LIN {X -15.999,Y -33.308,Z -148.499,A -90.000,B 90.000,C 0.000} C_DIS
LIN {X -18.536,Y -33.308,Z -146.844,A -90.000,B 90.000,C 0.000} C_DIS
LIN {X -19.606,Y -33.308,Z -146.164,A -90.000,B 90.000,C 0.000} C_DIS
LIN {X -20.856,Y -33.308,Z -145.200,A -90.000,B 90.000,C 0.000} C_DIS
LIN {X -22.809,Y -33.308,Z -143.742,A -90.000,B 90.000,C 0.000} C_DIS
LIN {X -23.151,Y -33.308,Z -143.479,A -90.000,B 90.000,C 0.000} C_DIS
LIN {X -23.524,Y -33.308,Z -143.181,A -90.000,B 90.000,C 0.000} C_DIS
LIN {X -25.307,Y -33.308,Z -141.556,A -90.000,B 90.000,C 0.000} C_DIS
LIN {X -26.828,Y -33.308,Z -140.210,A -90.000,B 90.000,C 0.000} C_DIS
LIN {X -27.168,Y -33.308,Z -139.876,A -90.000,B 90.000,C 0.000} C_DIS
LIN {X -27.524,Y -33.308,Z -139.495,A -90.000,B 90.000,C 0.000} C_DIS
LIN {X -28.033,Y -33.308,Z -138.967,A -90.000,B 90.000,C 0.000} C_DIS
LIN {X -30.108,Y -33.308,Z -136.726,A -90.000,B 90.000,C 0.000} C_DIS
LIN {X -30.362,Y -33.308,Z -136.404,A -90.000,B 90.000,C 0.000} C_DIS
LIN {X -31.175,Y -33.308,Z -135.330,A -90.000,B 90.000,C 0.000} C_DIS
LIN {X -32.732,Y -33.308,Z -133.288,A -90.000,B 90.000,C 0.000} C_DIS
LIN {X -32.993,Y -33.308,Z -132.891,A -90.000,B 90.000,C 0.000} C_DIS
LIN {X -34.951,Y -33.308,Z -129.675,A -90.000,B 90.000,C 0.000} C_DIS
LIN {X -35.160,Y -33.308,Z -129.243,A -90.000,B 90.000,C 0.000} C_DIS
LIN {X -36.562,Y -33.308,Z -126.281,A -90.000,B 90.000,C 0.000} C_DIS
LIN {X -36.636,Y -33.308,Z -126.118,A -90.000,B 90.000,C 0.000} C_DIS
LIN {X -37.764,Y -33.308,Z -123.048,A -90.000,B 90.000,C 0.000} C_DIS
LIN {X -37.875,Y -33.308,Z -122.732,A -90.000,B 90.000,C 0.000} C_DIS
LIN {X -37.915,Y -33.308,Z -122.610,A -90.000,B 90.000,C 0.000} C_DIS
LIN {X -38.201,Y -33.308,Z -121.561,A -90.000,B 90.000,C 0.000} C_DIS
LIN {X -38.605,Y -33.308,Z -120.049,A -90.000,B 90.000,C 0.000} C_DIS
LIN {X -38.751,Y -33.308,Z -119.515,A -90.000,B 90.000,C 0.000} C_DIS
LIN {X -38.857,Y -33.308,Z -119.060,A -90.000,B 90.000,C 0.000} C_DIS
LIN {X -39.050,Y -33.308,Z -118.006,A -90.000,B 90.000,C 0.000} C_DIS
LIN {X -39.335,Y -33.308,Z -116.504,A -90.000,B 90.000,C 0.000} C_DIS
LIN {X -39.510,Y -33.308,Z -115.571,A -90.000,B 90.000,C 0.000} C_DIS
LIN {X -39.533,Y -33.308,Z -115.382,A -90.000,B 90.000,C 0.000} C_DIS
LIN {X -39.662,Y -33.308,Z -114.053,A -90.000,B 90.000,C 0.000} C_DIS
LIN {X -39.769,Y -33.308,Z -112.841,A -90.000,B 90.000,C 0.000} C_DIS
LIN {X -39.851,Y -33.308,Z -111.994,A -90.000,B 90.000,C 0.000} C_DIS
LIN {X -39.881,Y -33.308,Z -111.571,A -90.000,B 90.000,C 0.000} C_DIS
LIN {X -39.882,Y -33.308,Z -111.344,A -90.000,B 90.000,C 0.000} C_DIS
LIN {X -39.887,Y -33.308,Z -111.029,A -90.000,B 90.000,C 0.000} C_DIS
LIN {X -39.893,Y -33.308,Z -109.551,A -90.000,B 90.000,C 0.000} C_DIS
LIN {X -39.909,Y -33.308,Z -108.367,A -90.000,B 90.000,C 0.000} C_DIS
LIN {X -39.903,Y -33.308,Z -107.912,A -90.000,B 90.000,C 0.000} C_DIS
LIN {X -39.874,Y -33.308,Z -107.539,A -90.000,B 90.000,C 0.000} C_DIS
LIN {X -39.834,Y -33.308,Z -106.670,A -90.000,B 90.000,C 0.000} C_DIS
LIN {X -39.843,Y -33.308,Z -106.632,A -90.000,B 90.000,C 0.000} C_DIS
LIN {X -40.216,Y -33.308,Z -105.871,A -90.000,B 90.000,C 0.000} C_DIS
LIN {X -40.541,Y -33.308,Z -105.425,A -90.000,B 90.000,C 0.000} C_DIS
LIN {X -41.279,Y -33.308,Z -104.304,A -90.000,B 90.000,C 0.000} C_DIS
LIN {X -41.681,Y -33.308,Z -103.742,A -90.000,B 90.000,C 0.000} C_DIS
LIN {X -42.580,Y -33.308,Z -102.613,A -90.000,B 90.000,C 0.000} C_DIS
LIN {X -42.846,Y -33.308,Z -102.253,A -90.000,B 90.000,C 0.000} C_DIS
LIN {X -43.563,Y -33.308,Z -101.346,A -90.000,B 90.000,C 0.000} C_DIS
LIN {X -44.397,Y -33.308,Z -100.200,A -90.000,B 90.000,C 0.000} C_DIS
LIN {X -44.716,Y -33.308,Z -99.731,A -90.000,B 90.000,C 0.000} C_DIS
LIN {X -45.686,Y -33.308,Z -98.284,A -90.000,B 90.000,C 0.000} C_DIS
LIN {X -46.185,Y -33.308,Z -97.544,A -90.000,B 90.000,C 0.000} C_DIS
LIN {X -46.405,Y -33.308,Z -97.201,A -90.000,B 90.000,C 0.000} C_DIS
LIN {X -46.712,Y -33.308,Z -96.706,A -90.000,B 90.000,C 0.000} C_DIS
LIN {X -47.443,Y -33.308,Z -95.513,A -90.000,B 90.000,C 0.000} C_DIS
LIN {X -47.884,Y -33.308,Z -94.789,A -90.000,B 90.000,C 0.000} C_DIS
LIN {X -48.028,Y -33.308,Z -94.546,A -90.000,B 90.000,C 0.000} C_DIS
LIN {X -48.144,Y -33.308,Z -94.332,A -90.000,B 90.000,C 0.000} C_DIS
LIN {X -48.227,Y -33.308,Z -94.169,A -90.000,B 90.000,C 0.000} C_DIS
LIN {X -49.715,Y -33.308,Z -90.825,A -90.000,B 90.000,C 0.000} C_DIS
LIN {X -49.898,Y -33.308,Z -90.362,A -90.000,B 90.000,C 0.000} C_DIS
LIN {X -50.066,Y -33.308,Z -89.882,A -90.000,B 90.000,C 0.000} C_DIS
LIN {X -50.156,Y -33.308,Z -89.607,A -90.000,B 90.000,C 0.000} C_DIS
LIN {X -50.572,Y -33.308,Z -88.253,A -90.000,B 90.000,C 0.000} C_DIS
LIN {X -50.836,Y -33.308,Z -87.423,A -90.000,B 90.000,C 0.000} C_DIS
LIN {X -51.046,Y -33.308,Z -86.747,A -90.000,B 90.000,C 0.000} C_DIS
LIN {X -51.153,Y -33.308,Z -86.380,A -90.000,B 90.000,C 0.000} C_DIS
LIN {X -51.746,Y -33.308,Z -84.240,A -90.000,B 90.000,C 0.000} C_DIS
LIN {X -52.221,Y -33.308,Z -82.065,A -90.000,B 90.000,C 0.000} C_DIS
LIN {X -52.576,Y -33.308,Z -80.127,A -90.000,B 90.000,C 0.000} C_DIS
LIN {X -52.615,Y -33.308,Z -79.847,A -90.000,B 90.000,C 0.000} C_DIS
LIN {X -52.708,Y -33.308,Z -78.854,A -90.000,B 90.000,C 0.000} C_DIS
LIN {X -52.791,Y -33.308,Z -78.084,A -90.000,B 90.000,C 0.000} C_DIS
LIN {X -52.824,Y -33.308,Z -76.672,A -90.000,B 90.000,C 0.000} C_DIS
LIN {X -52.824,Y -33.308,Z -76.379,A -90.000,B 90.000,C 0.000} C_DIS
LIN {X -52.821,Y -33.308,Z -76.293,A -90.000,B 90.000,C 0.000} C_DIS
LIN {X -52.840,Y -33.308,Z -76.082,A -90.000,B 90.000,C 0.000} C_DIS
LIN {X -52.839,Y -33.308,Z -74.765,A -90.000,B 90.000,C 0.000} C_DIS
LIN {X -52.858,Y -33.308,Z -74.482,A -90.000,B 90.000,C 0.000} C_DIS
LIN {X -52.768,Y -33.308,Z -73.356,A -90.000,B 90.000,C 0.000} C_DIS
LIN {X -52.777,Y -33.308,Z -72.948,A -90.000,B 90.000,C 0.000} C_DIS
LIN {X -52.757,Y -33.308,Z -72.712,A -90.000,B 90.000,C 0.000} C_DIS
LIN {X -52.602,Y -33.308,Z -71.811,A -90.000,B 90.000,C 0.000} C_DIS
LIN {X -52.589,Y -33.308,Z -71.493,A -90.000,B 90.000,C 0.000} C_DIS
LIN {X -52.569,Y -33.308,Z -71.257,A -90.000,B 90.000,C 0.000} C_DIS
LIN {X -52.319,Y -33.308,Z -70.370,A -90.000,B 90.000,C 0.000} C_DIS
LIN {X -52.254,Y -33.308,Z -69.902,A -90.000,B 90.000,C 0.000} C_DIS
LIN {X -52.185,Y -33.308,Z -69.675,A -90.000,B 90.000,C 0.000} C_DIS
LIN {X -51.762,Y -33.308,Z -68.858,A -90.000,B 90.000,C 0.000} C_DIS
LIN {X -51.636,Y -33.308,Z -68.514,A -90.000,B 90.000,C 0.000} C_DIS
LIN {X -51.589,Y -33.308,Z -68.423,A -90.000,B 90.000,C 0.000} C_DIS
LIN {X -51.480,Y -33.308,Z -68.226,A -90.000,B 90.000,C 0.000} C_DIS
LIN {X -51.476,Y -33.308,Z -68.222,A -90.000,B 90.000,C 0.000} C_DIS
LIN {X -51.325,Y -33.308,Z -68.048,A -90.000,B 90.000,C 0.000} C_DIS
LIN {X -50.280,Y -33.308,Z -66.958,A -90.000,B 90.000,C 0.000} C_DIS
LIN {X -50.251,Y -33.308,Z -66.924,A -90.000,B 90.000,C 0.000} C_DIS
LIN {X -50.061,Y -33.308,Z -66.782,A -90.000,B 90.000,C 0.000} C_DIS
LIN {X -50.009,Y -33.308,Z -66.752,A -90.000,B 90.000,C 0.000} C_DIS
LIN {X -49.012,Y -33.308,Z -66.062,A -90.000,B 90.000,C 0.000} C_DIS
LIN {X -48.527,Y -33.308,Z -65.766,A -90.000,B 90.000,C 0.000} C_DIS
LIN {X -48.102,Y -33.308,Z -65.546,A -90.000,B 90.000,C 0.000} C_DIS
LIN {X -47.850,Y -33.308,Z -65.419,A -90.000,B 90.000,C 0.000} C_DIS
LIN {X -46.602,Y -33.308,Z -64.968,A -90.000,B 90.000,C 0.000} C_DIS
LIN {X -45.421,Y -33.308,Z -64.531,A -90.000,B 90.000,C 0.000} C_DIS
LIN {X -45.151,Y -33.308,Z -64.451,A -90.000,B 90.000,C 0.000} C_DIS
LIN {X -44.503,Y -33.308,Z -64.272,A -90.000,B 90.000,C 0.000} C_DIS
LIN {X -43.209,Y -33.308,Z -63.965,A -90.000,B 90.000,C 0.000} C_DIS
LIN {X -43.095,Y -33.308,Z -63.939,A -90.000,B 90.000,C 0.000} C_DIS
LIN {X -40.860,Y -33.308,Z -63.512,A -90.000,B 90.000,C 0.000} C_DIS
LIN {X -40.000,Y -33.308,Z -63.408,A -90.000,B 90.000,C 0.000} C_DIS
LIN {X -39.681,Y -33.308,Z -63.385,A -90.000,B 90.000,C 0.000} C_DIS
LIN {X -39.254,Y -33.308,Z -63.373,A -90.000,B 90.000,C 0.000} C_DIS
LIN {X -36.732,Y -33.308,Z -63.251,A -90.000,B 90.000,C 0.000} C_DIS
LIN {X -35.728,Y -33.308,Z -63.273,A -90.000,B 90.000,C 0.000} C_DIS
LIN {X -35.378,Y -33.308,Z -63.300,A -90.000,B 90.000,C 0.000} C_DIS
LIN {X -33.474,Y -33.308,Z -63.465,A -90.000,B 90.000,C 0.000} C_DIS
LIN {X -33.246,Y -33.308,Z -63.489,A -90.000,B 90.000,C 0.000} C_DIS
LIN {X -32.432,Y -33.308,Z -63.617,A -90.000,B 90.000,C 0.000} C_DIS
LIN {X -30.767,Y -33.308,Z -63.887,A -90.000,B 90.000,C 0.000} C_DIS
LIN {X -30.545,Y -33.308,Z -63.929,A -90.000,B 90.000,C 0.000} C_DIS
LIN {X -30.194,Y -33.308,Z -63.999,A -90.000,B 90.000,C 0.000} C_DIS
LIN {X -28.705,Y -33.308,Z -64.309,A -90.000,B 90.000,C 0.000} C_DIS
LIN {X -28.123,Y -33.308,Z -64.436,A -90.000,B 90.000,C 0.000} C_DIS
LIN {X -28.013,Y -33.308,Z -64.462,A -90.000,B 90.000,C 0.000} C_DIS
LIN {X -25.914,Y -33.308,Z -65.027,A -90.000,B 90.000,C 0.000} C_DIS
LIN {X -24.380,Y -33.308,Z -65.532,A -90.000,B 90.000,C 0.000} C_DIS
LIN {X -24.132,Y -33.308,Z -65.610,A -90.000,B 90.000,C 0.000} C_DIS
LIN {X -23.744,Y -33.308,Z -65.739,A -90.000,B 90.000,C 0.000} C_DIS
LIN {X -22.588,Y -33.308,Z -66.146,A -90.000,B 90.000,C 0.000} C_DIS
LIN {X -21.576,Y -33.308,Z -66.458,A -90.000,B 90.000,C 0.000} C_DIS
LIN {X -21.536,Y -33.308,Z -66.468,A -90.000,B 90.000,C 0.000} C_DIS
LIN {X -21.279,Y -33.308,Z -65.952,A -90.000,B 90.000,C 0.000} C_DIS
LIN {X -21.202,Y -33.308,Z -65.724,A -90.000,B 90.000,C 0.000} C_DIS
LIN {X -20.968,Y -33.308,Z -65.093,A -90.000,B 90.000,C 0.000} C_DIS
LIN {X -20.909,Y -33.308,Z -64.895,A -90.000,B 90.000,C 0.000} C_DIS
LIN {X -20.659,Y -33.308,Z -64.202,A -90.000,B 90.000,C 0.000} C_DIS
LIN {X -20.533,Y -33.308,Z -63.908,A -90.000,B 90.000,C 0.000} C_DIS
LIN {X -20.359,Y -33.308,Z -63.600,A -90.000,B 90.000,C 0.000} C_DIS
LIN {X -20.270,Y -33.308,Z -63.460,A -90.000,B 90.000,C 0.000} C_DIS
LIN {X -19.954,Y -33.308,Z -62.911,A -90.000,B 90.000,C 0.000} C_DIS
LIN {X -19.740,Y -33.308,Z -62.631,A -90.000,B 90.000,C 0.000} C_DIS
LIN {X -19.479,Y -33.308,Z -62.376,A -90.000,B 90.000,C 0.000} C_DIS
LIN {X -19.448,Y -33.308,Z -62.349,A -90.000,B 90.000,C 0.000} C_DIS
LIN {X -19.165,Y -33.308,Z -62.141,A -90.000,B 90.000,C 0.000} C_DIS
LIN {X -18.817,Y -33.308,Z -61.902,A -90.000,B 90.000,C 0.000} C_DIS
LIN {X -18.540,Y -33.308,Z -61.737,A -90.000,B 90.000,C 0.000} C_DIS
LIN {X -18.265,Y -33.308,Z -61.626,A -90.000,B 90.000,C 0.000} C_DIS
LIN {X -17.942,Y -33.308,Z -61.498,A -90.000,B 90.000,C 0.000} C_DIS
LIN {X -17.612,Y -33.308,Z -61.377,A -90.000,B 90.000,C 0.000} C_DIS
LIN {X -16.997,Y -33.308,Z -61.181,A -90.000,B 90.000,C 0.000} C_DIS
LIN {X -16.111,Y -33.308,Z -60.930,A -90.000,B 90.000,C 0.000} C_DIS
LIN {X -15.997,Y -33.308,Z -60.903,A -90.000,B 90.000,C 0.000} C_DIS
LIN {X -15.606,Y -33.308,Z -60.822,A -90.000,B 90.000,C 0.000} C_DIS
LIN {X -15.503,Y -33.308,Z -60.804,A -90.000,B 90.000,C 0.000} C_DIS
LIN {X -15.152,Y -33.308,Z -60.781,A -90.000,B 90.000,C 0.000} C_DIS
LIN {X -12.993,Y -33.308,Z -60.780,A -90.000,B 90.000,C 0.000} C_DIS
LIN {X -11.855,Y -33.308,Z -60.776,A -90.000,B 90.000,C 0.000} C_DIS
LIN {X -11.504,Y -33.308,Z -60.803,A -90.000,B 90.000,C 0.000} C_DIS
LIN {X -11.122,Y -33.308,Z -60.840,A -90.000,B 90.000,C 0.000} C_DIS
LIN {X -8.836,Y -33.308,Z -61.073,A -90.000,B 90.000,C 0.000} C_DIS
LIN {X -7.942,Y -33.308,Z -61.208,A -90.000,B 90.000,C 0.000} C_DIS
LIN {X -6.167,Y -33.308,Z -61.448,A -90.000,B 90.000,C 0.000} C_DIS
LIN {X -5.366,Y -33.308,Z -61.575,A -90.000,B 90.000,C 0.000} C_DIS
LIN {X -4.569,Y -33.308,Z -61.716,A -90.000,B 90.000,C 0.000} C_DIS
LIN {X -2.737,Y -33.308,Z -61.952,A -90.000,B 90.000,C 0.000} C_DIS
LIN {X -1.013,Y -33.308,Z -62.234,A -90.000,B 90.000,C 0.000} C_DIS
LIN {X 0.927,Y -33.308,Z -62.435,A -90.000,B 90.000,C 0.000} C_DIS
LIN {X 1.948,Y -33.308,Z -62.549,A -90.000,B 90.000,C 0.000} C_DIS
LIN {X 2.990,Y -33.308,Z -62.617,A -90.000,B 90.000,C 0.000} C_DIS
LIN {X 4.660,Y -33.308,Z -62.776,A -90.000,B 90.000,C 0.000} C_DIS
LIN {X 5.580,Y -33.308,Z -62.844,A -90.000,B 90.000,C 0.000} C_DIS
LIN {X 6.790,Y -33.308,Z -62.924,A -90.000,B 90.000,C 0.000} C_DIS
LIN {X 7.569,Y -33.308,Z -62.950,A -90.000,B 90.000,C 0.000} C_DIS
LIN {X 8.530,Y -33.308,Z -62.986,A -90.000,B 90.000,C 0.000} C_DIS
LIN {X 9.844,Y -33.308,Z -62.969,A -90.000,B 90.000,C 0.000} C_DIS
LIN {X 10.732,Y -33.308,Z -62.896,A -90.000,B 90.000,C 0.000} C_DIS
LIN {X 11.400,Y -33.308,Z -62.776,A -90.000,B 90.000,C 0.000} C_DIS
LIN {X 11.835,Y -33.308,Z -62.634,A -90.000,B 90.000,C 0.000} C_DIS
LIN {X 12.131,Y -33.308,Z -62.482,A -90.000,B 90.000,C 0.000} C_DIS
LIN {X 12.597,Y -33.308,Z -62.206,A -90.000,B 90.000,C 0.000} C_DIS
LIN {X 12.961,Y -33.308,Z -62.010,A -90.000,B 90.000,C 0.000} C_DIS
LIN {X 13.229,Y -33.308,Z -61.872,A -90.000,B 90.000,C 0.000} C_DIS
LIN {X 13.616,Y -33.308,Z -61.666,A -90.000,B 90.000,C 0.000} C_DIS
LIN {X 13.852,Y -33.308,Z -61.563,A -90.000,B 90.000,C 0.000} C_DIS
LIN {X 14.231,Y -33.308,Z -61.424,A -90.000,B 90.000,C 0.000} C_DIS
LIN {X 14.576,Y -33.308,Z -61.333,A -90.000,B 90.000,C 0.000} C_DIS
LIN {X 14.698,Y -33.308,Z -61.293,A -90.000,B 90.000,C 0.000} C_DIS
LIN {X 14.742,Y -33.308,Z -61.279,A -90.000,B 90.000,C 0.000} C_DIS
LIN {X 14.860,Y -33.308,Z -61.243,A -90.000,B 90.000,C 0.000} C_DIS
LIN {X 15.253,Y -33.308,Z -61.152,A -90.000,B 90.000,C 0.000} C_DIS
LIN {X 15.653,Y -33.308,Z -61.110,A -90.000,B 90.000,C 0.000} C_DIS
LIN {X 15.830,Y -33.308,Z -61.103,A -90.000,B 90.000,C 0.000} C_DIS
LIN {X 16.705,Y -33.308,Z -61.121,A -90.000,B 90.000,C 0.000} C_DIS
LIN {X 17.110,Y -33.308,Z -61.177,A -90.000,B 90.000,C 0.000} C_DIS
LIN {X 17.392,Y -33.308,Z -61.217,A -90.000,B 90.000,C 0.000} C_DIS
LIN {X 17.618,Y -33.308,Z -61.255,A -90.000,B 90.000,C 0.000} C_DIS
LIN {X 17.736,Y -33.308,Z -61.278,A -90.000,B 90.000,C 0.000} C_DIS
LIN {X 17.944,Y -33.308,Z -61.166,A -90.000,B 90.000,C 0.000} C_DIS
LIN {X 18.039,Y -33.308,Z -61.122,A -90.000,B 90.000,C 0.000} C_DIS
LIN {X 18.354,Y -33.308,Z -60.997,A -90.000,B 90.000,C 0.000} C_DIS
LIN {X 18.590,Y -33.308,Z -60.833,A -90.000,B 90.000,C 0.000} C_DIS
LIN {X 18.755,Y -33.308,Z -60.737,A -90.000,B 90.000,C 0.000} C_DIS
LIN {X 18.966,Y -33.308,Z -60.623,A -90.000,B 90.000,C 0.000} C_DIS
LIN {X 19.141,Y -33.308,Z -60.546,A -90.000,B 90.000,C 0.000} C_DIS
LIN {X 19.364,Y -33.308,Z -60.457,A -90.000,B 90.000,C 0.000} C_DIS
LIN {X 19.546,Y -33.308,Z -60.401,A -90.000,B 90.000,C 0.000} C_DIS
LIN {X 19.884,Y -33.308,Z -60.310,A -90.000,B 90.000,C 0.000} C_DIS
LIN {X 20.034,Y -33.308,Z -60.279,A -90.000,B 90.000,C 0.000} C_DIS
LIN {X 20.311,Y -33.308,Z -60.238,A -90.000,B 90.000,C 0.000} C_DIS
LIN {X 20.453,Y -33.308,Z -60.219,A -90.000,B 90.000,C 0.000} C_DIS
LIN {X 20.876,Y -33.308,Z -60.209,A -90.000,B 90.000,C 0.000} C_DIS
LIN {X 21.298,Y -33.308,Z -60.250,A -90.000,B 90.000,C 0.000} C_DIS
LIN {X 21.856,Y -33.308,Z -60.371,A -90.000,B 90.000,C 0.000} C_DIS
LIN {X 22.005,Y -33.308,Z -60.420,A -90.000,B 90.000,C 0.000} C_DIS
LIN {X 22.223,Y -33.308,Z -60.253,A -90.000,B 90.000,C 0.000} C_DIS
LIN {X 22.475,Y -33.308,Z -60.067,A -90.000,B 90.000,C 0.000} C_DIS
LIN {X 22.603,Y -33.308,Z -59.979,A -90.000,B 90.000,C 0.000} C_DIS
LIN {X 22.940,Y -33.308,Z -59.756,A -90.000,B 90.000,C 0.000} C_DIS
LIN {X 23.193,Y -33.308,Z -59.603,A -90.000,B 90.000,C 0.000} C_DIS
LIN {X 23.466,Y -33.308,Z -59.442,A -90.000,B 90.000,C 0.000} C_DIS
LIN {X 23.667,Y -33.308,Z -59.330,A -90.000,B 90.000,C 0.000} C_DIS
LIN {X 24.032,Y -33.308,Z -59.140,A -90.000,B 90.000,C 0.000} C_DIS
LIN {X 24.416,Y -33.308,Z -58.965,A -90.000,B 90.000,C 0.000} C_DIS
LIN {X 24.819,Y -33.308,Z -58.788,A -90.000,B 90.000,C 0.000} C_DIS
LIN {X 25.037,Y -33.308,Z -58.701,A -90.000,B 90.000,C 0.000} C_DIS
LIN {X 25.238,Y -33.308,Z -58.623,A -90.000,B 90.000,C 0.000} C_DIS
LIN {X 25.658,Y -33.308,Z -58.481,A -90.000,B 90.000,C 0.000} C_DIS
LIN {X 25.742,Y -33.308,Z -58.455,A -90.000,B 90.000,C 0.000} C_DIS
LIN {X 25.705,Y -33.308,Z -58.141,A -90.000,B 90.000,C 0.000} C_DIS
LIN {X 25.684,Y -33.308,Z -57.920,A -90.000,B 90.000,C 0.000} C_DIS
LIN {X 25.655,Y -33.308,Z -57.445,A -90.000,B 90.000,C 0.000} C_DIS
LIN {X 25.677,Y -33.308,Z -56.969,A -90.000,B 90.000,C 0.000} C_DIS
LIN {X 25.730,Y -33.308,Z -56.579,A -90.000,B 90.000,C 0.000} C_DIS
LIN {X 25.823,Y -33.308,Z -56.121,A -90.000,B 90.000,C 0.000} C_DIS
LIN {X 25.964,Y -33.308,Z -55.675,A -90.000,B 90.000,C 0.000} C_DIS
LIN {X 26.151,Y -33.308,Z -55.247,A -90.000,B 90.000,C 0.000} C_DIS
LIN {X 26.465,Y -33.308,Z -54.700,A -90.000,B 90.000,C 0.000} C_DIS
LIN {X 26.502,Y -33.308,Z -54.645,A -90.000,B 90.000,C 0.000} C_DIS
LIN {X 26.706,Y -33.308,Z -54.362,A -90.000,B 90.000,C 0.000} C_DIS
LIN {X 26.778,Y -33.308,Z -54.272,A -90.000,B 90.000,C 0.000} C_DIS
LIN {X 27.012,Y -33.308,Z -54.013,A -90.000,B 90.000,C 0.000} C_DIS
LIN {X 27.093,Y -33.308,Z -53.931,A -90.000,B 90.000,C 0.000} C_DIS
LIN {X 27.353,Y -33.308,Z -53.699,A -90.000,B 90.000,C 0.000} C_DIS
LIN {X 27.443,Y -33.308,Z -53.626,A -90.000,B 90.000,C 0.000} C_DIS
LIN {X 27.726,Y -33.308,Z -53.423,A -90.000,B 90.000,C 0.000} C_DIS
LIN {X 27.823,Y -33.308,Z -53.360,A -90.000,B 90.000,C 0.000} C_DIS
LIN {X 28.127,Y -33.308,Z -53.188,A -90.000,B 90.000,C 0.000} C_DIS
LIN {X 28.289,Y -33.308,Z -53.103,A -90.000,B 90.000,C 0.000} C_DIS
LIN {X 28.423,Y -33.308,Z -53.037,A -90.000,B 90.000,C 0.000} C_DIS
LIN {X 28.711,Y -33.308,Z -52.912,A -90.000,B 90.000,C 0.000} C_DIS
LIN {X 28.851,Y -33.308,Z -52.861,A -90.000,B 90.000,C 0.000} C_DIS
LIN {X 29.151,Y -33.308,Z -52.767,A -90.000,B 90.000,C 0.000} C_DIS
LIN {X 29.219,Y -33.308,Z -52.748,A -90.000,B 90.000,C 0.000} C_DIS
LIN {X 29.223,Y -33.308,Z -52.612,A -90.000,B 90.000,C 0.000} C_DIS
LIN {X 29.286,Y -33.308,Z -52.163,A -90.000,B 90.000,C 0.000} C_DIS
LIN {X 29.356,Y -33.308,Z -51.864,A -90.000,B 90.000,C 0.000} C_DIS
LIN {X 29.424,Y -33.308,Z -51.550,A -90.000,B 90.000,C 0.000} C_DIS
LIN {X 29.529,Y -33.308,Z -51.140,A -90.000,B 90.000,C 0.000} C_DIS
LIN {X 29.681,Y -33.308,Z -50.745,A -90.000,B 90.000,C 0.000} C_DIS
LIN {X 29.756,Y -33.308,Z -50.567,A -90.000,B 90.000,C 0.000} C_DIS
LIN {X 29.940,Y -33.308,Z -50.168,A -90.000,B 90.000,C 0.000} C_DIS
LIN {X 30.138,Y -33.308,Z -49.793,A -90.000,B 90.000,C 0.000} C_DIS
LIN {X 30.158,Y -33.308,Z -49.758,A -90.000,B 90.000,C 0.000} C_DIS
LIN {X 30.387,Y -33.308,Z -49.416,A -90.000,B 90.000,C 0.000} C_DIS
LIN {X 30.427,Y -33.308,Z -49.361,A -90.000,B 90.000,C 0.000} C_DIS
LIN {X 30.699,Y -33.308,Z -48.997,A -90.000,B 90.000,C 0.000} C_DIS
LIN {X 30.764,Y -33.308,Z -48.903,A -90.000,B 90.000,C 0.000} C_DIS
LIN {X 30.798,Y -33.308,Z -48.858,A -90.000,B 90.000,C 0.000} C_DIS
LIN {X 31.083,Y -33.308,Z -48.522,A -90.000,B 90.000,C 0.000} C_DIS
LIN {X 31.405,Y -33.308,Z -48.220,A -90.000,B 90.000,C 0.000} C_DIS
LIN {X 31.941,Y -33.308,Z -47.791,A -90.000,B 90.000,C 0.000} C_DIS
LIN {X 31.970,Y -33.308,Z -47.764,A -90.000,B 90.000,C 0.000} C_DIS
LIN {X 32.324,Y -33.308,Z -47.500,A -90.000,B 90.000,C 0.000} C_DIS
LIN {X 32.717,Y -33.308,Z -47.272,A -90.000,B 90.000,C 0.000} C_DIS
LIN {X 32.794,Y -33.308,Z -47.233,A -90.000,B 90.000,C 0.000} C_DIS
LIN {X 33.121,Y -33.308,Z -47.090,A -90.000,B 90.000,C 0.000} C_DIS
LIN {X 33.449,Y -33.308,Z -46.955,A -90.000,B 90.000,C 0.000} C_DIS
LIN {X 33.884,Y -33.308,Z -46.784,A -90.000,B 90.000,C 0.000} C_DIS
LIN {X 34.311,Y -33.308,Z -46.652,A -90.000,B 90.000,C 0.000} C_DIS
LIN {X 34.813,Y -33.308,Z -46.529,A -90.000,B 90.000,C 0.000} C_DIS
LIN {X 35.264,Y -33.308,Z -46.469,A -90.000,B 90.000,C 0.000} C_DIS
LIN {X 35.688,Y -33.308,Z -46.434,A -90.000,B 90.000,C 0.000} C_DIS
LIN {X 36.302,Y -33.308,Z -46.365,A -90.000,B 90.000,C 0.000} C_DIS
LIN {X 36.835,Y -33.308,Z -46.338,A -90.000,B 90.000,C 0.000} C_DIS
LIN {X 37.302,Y -33.308,Z -46.347,A -90.000,B 90.000,C 0.000} C_DIS
LIN {X 37.688,Y -33.308,Z -46.382,A -90.000,B 90.000,C 0.000} C_DIS
LIN {X 38.275,Y -33.308,Z -46.449,A -90.000,B 90.000,C 0.000} C_DIS
LIN {X 38.738,Y -33.308,Z -46.508,A -90.000,B 90.000,C 0.000} C_DIS
LIN {X 39.091,Y -33.308,Z -46.568,A -90.000,B 90.000,C 0.000} C_DIS
LIN {X 40.567,Y -33.308,Z -46.891,A -90.000,B 90.000,C 0.000} C_DIS
LIN {X 41.529,Y -33.308,Z -47.060,A -90.000,B 90.000,C 0.000} C_DIS
LIN {X 42.172,Y -33.308,Z -47.093,A -90.000,B 90.000,C 0.000} C_DIS
LIN {X 43.024,Y -33.308,Z -46.949,A -90.000,B 90.000,C 0.000} C_DIS
LIN {X 43.517,Y -33.308,Z -46.826,A -90.000,B 90.000,C 0.000} C_DIS
LIN {X 44.454,Y -33.308,Z -46.576,A -90.000,B 90.000,C 0.000} C_DIS
LIN {X 45.621,Y -33.308,Z -46.357,A -90.000,B 90.000,C 0.000} C_DIS
LIN {X 46.224,Y -33.308,Z -46.219,A -90.000,B 90.000,C 0.000} C_DIS
LIN {X 46.763,Y -33.308,Z -46.136,A -90.000,B 90.000,C 0.000} C_DIS
LIN {X 47.215,Y -33.308,Z -46.104,A -90.000,B 90.000,C 0.000} C_DIS
LIN {X 47.811,Y -33.308,Z -46.089,A -90.000,B 90.000,C 0.000} C_DIS
LIN {X 48.729,Y -33.308,Z -46.110,A -90.000,B 90.000,C 0.000} C_DIS
LIN {X 49.207,Y -33.308,Z -46.147,A -90.000,B 90.000,C 0.000} C_DIS
LIN {X 49.600,Y -33.308,Z -46.184,A -90.000,B 90.000,C 0.000} C_DIS
LIN {X 50.226,Y -33.308,Z -46.292,A -90.000,B 90.000,C 0.000} C_DIS
LIN {X 50.651,Y -33.308,Z -46.408,A -90.000,B 90.000,C 0.000} C_DIS
LIN {X 51.282,Y -33.308,Z -46.611,A -90.000,B 90.000,C 0.000} C_DIS
LIN {X 52.189,Y -33.308,Z -46.925,A -90.000,B 90.000,C 0.000} C_DIS
LIN {X 53.231,Y -33.308,Z -47.364,A -90.000,B 90.000,C 0.000} C_DIS
LIN {X 53.647,Y -33.308,Z -47.549,A -90.000,B 90.000,C 0.000} C_DIS
LIN {X 54.040,Y -33.308,Z -47.779,A -90.000,B 90.000,C 0.000} C_DIS
LIN {X 56.196,Y -33.308,Z -49.211,A -90.000,B 90.000,C 0.000} C_DIS
LIN {X 56.730,Y -33.308,Z -49.569,A -90.000,B 90.000,C 0.000} C_DIS
LIN {X 57.096,Y -33.308,Z -49.840,A -90.000,B 90.000,C 0.000} C_DIS
LIN {X 59.476,Y -33.308,Z -51.862,A -90.000,B 90.000,C 0.000} C_DIS
LIN {X 59.810,Y -33.308,Z -52.171,A -90.000,B 90.000,C 0.000} C_DIS
LIN {X 62.039,Y -33.308,Z -54.281,A -90.000,B 90.000,C 0.000} C_DIS
LIN {X 63.618,Y -33.308,Z -55.808,A -90.000,B 90.000,C 0.000} C_DIS
LIN {X 64.198,Y -33.308,Z -56.378,A -90.000,B 90.000,C 0.000} C_DIS
LIN {X 64.715,Y -33.308,Z -56.862,A -90.000,B 90.000,C 0.000} C_DIS
LIN {X 66.205,Y -33.308,Z -58.228,A -90.000,B 90.000,C 0.000} C_DIS
LIN {X 68.301,Y -33.308,Z -60.193,A -90.000,B 90.000,C 0.000} C_DIS
LIN {X 69.366,Y -33.308,Z -61.311,A -90.000,B 90.000,C 0.000} C_DIS
LIN {X 70.233,Y -33.308,Z -62.330,A -90.000,B 90.000,C 0.000} C_DIS
LIN {X 71.735,Y -33.308,Z -64.192,A -90.000,B 90.000,C 0.000} C_DIS
LIN {X 71.839,Y -33.308,Z -64.323,A -90.000,B 90.000,C 0.000} C_DIS
LIN {X 72.046,Y -33.308,Z -64.596,A -90.000,B 90.000,C 0.000} C_DIS
LIN {X 72.489,Y -33.308,Z -65.199,A -90.000,B 90.000,C 0.000} C_DIS
LIN {X 72.909,Y -33.308,Z -65.812,A -90.000,B 90.000,C 0.000} C_DIS
LIN {X 73.188,Y -33.308,Z -66.158,A -90.000,B 90.000,C 0.000} C_DIS
LIN {X 73.389,Y -33.308,Z -66.438,A -90.000,B 90.000,C 0.000} C_DIS
LIN {X 73.517,Y -33.308,Z -66.628,A -90.000,B 90.000,C 0.000} C_DIS
LIN {X 73.829,Y -33.308,Z -67.008,A -90.000,B 90.000,C 0.000} C_DIS
LIN {X 74.218,Y -33.308,Z -67.509,A -90.000,B 90.000,C 0.000} C_DIS
LIN {X 74.278,Y -33.308,Z -67.577,A -90.000,B 90.000,C 0.000} C_DIS
LIN {X 74.534,Y -33.308,Z -67.914,A -90.000,B 90.000,C 0.000} C_DIS
LIN {X 74.861,Y -33.308,Z -68.353,A -90.000,B 90.000,C 0.000} C_DIS
LIN {X 75.321,Y -33.308,Z -68.845,A -90.000,B 90.000,C 0.000} C_DIS
LIN {X 75.520,Y -33.308,Z -69.107,A -90.000,B 90.000,C 0.000} C_DIS
LIN {X 76.204,Y -33.308,Z -69.865,A -90.000,B 90.000,C 0.000} C_DIS
LIN {X 76.275,Y -33.308,Z -69.948,A -90.000,B 90.000,C 0.000} C_DIS
LIN {X 76.321,Y -33.308,Z -69.996,A -90.000,B 90.000,C 0.000} C_DIS
LIN {X 76.568,Y -33.308,Z -70.298,A -90.000,B 90.000,C 0.000} C_DIS
LIN {X 76.871,Y -33.308,Z -70.672,A -90.000,B 90.000,C 0.000} C_DIS
LIN {X 77.245,Y -33.308,Z -71.078,A -90.000,B 90.000,C 0.000} C_DIS
LIN {X 77.541,Y -33.308,Z -71.404,A -90.000,B 90.000,C 0.000} C_DIS
LIN {X 77.612,Y -33.308,Z -71.491,A -90.000,B 90.000,C 0.000} C_DIS
LIN {X 77.796,Y -33.308,Z -71.699,A -90.000,B 90.000,C 0.000} C_DIS
LIN {X 78.092,Y -33.308,Z -72.049,A -90.000,B 90.000,C 0.000} C_DIS
LIN {X 78.123,Y -33.308,Z -71.941,A -90.000,B 90.000,C 0.000} C_DIS
LIN {X 78.695,Y -33.308,Z -70.203,A -90.000,B 90.000,C 0.000} C_DIS
LIN {X 78.831,Y -33.308,Z -69.802,A -90.000,B 90.000,C 0.000} C_DIS
LIN {X 79.195,Y -33.308,Z -68.754,A -90.000,B 90.000,C 0.000} C_DIS
LIN {X 79.783,Y -33.308,Z -67.276,A -90.000,B 90.000,C 0.000} C_DIS
LIN {X 79.809,Y -33.308,Z -67.218,A -90.000,B 90.000,C 0.000} C_DIS
LIN {X 80.447,Y -33.308,Z -65.768,A -90.000,B 90.000,C 0.000} C_DIS
LIN {X 80.647,Y -33.308,Z -65.330,A -90.000,B 90.000,C 0.000} C_DIS
LIN {X 81.438,Y -33.308,Z -63.804,A -90.000,B 90.000,C 0.000} C_DIS
LIN {X 81.684,Y -33.308,Z -63.383,A -90.000,B 90.000,C 0.000} C_DIS
LIN {X 82.705,Y -33.308,Z -61.742,A -90.000,B 90.000,C 0.000} C_DIS
LIN {X 84.243,Y -33.308,Z -59.630,A -90.000,B 90.000,C 0.000} C_DIS
LIN {X 85.732,Y -33.308,Z -57.856,A -90.000,B 90.000,C 0.000} C_DIS
LIN {X 86.059,Y -33.308,Z -57.494,A -90.000,B 90.000,C 0.000} C_DIS
LIN {X 87.795,Y -33.308,Z -55.685,A -90.000,B 90.000,C 0.000} C_DIS
LIN {X 89.787,Y -33.308,Z -53.862,A -90.000,B 90.000,C 0.000} C_DIS
LIN {X 90.167,Y -33.308,Z -53.520,A -90.000,B 90.000,C 0.000} C_DIS
LIN {X 92.263,Y -33.308,Z -51.722,A -90.000,B 90.000,C 0.000} C_DIS
LIN {X 94.367,Y -33.308,Z -49.945,A -90.000,B 90.000,C 0.000} C_DIS
LIN {X 94.745,Y -33.308,Z -49.614,A -90.000,B 90.000,C 0.000} C_DIS
LIN {X 94.732,Y -33.308,Z -49.589,A -90.000,B 90.000,C 0.000} C_DIS
LIN {X 94.667,Y -33.308,Z -49.441,A -90.000,B 90.000,C 0.000} C_DIS
LIN {X 94.423,Y -33.308,Z -48.996,A -90.000,B 90.000,C 0.000} C_DIS
LIN {X 94.322,Y -33.308,Z -48.808,A -90.000,B 90.000,C 0.000} C_DIS
LIN {X 94.232,Y -33.308,Z -48.623,A -90.000,B 90.000,C 0.000} C_DIS
LIN {X 94.145,Y -33.308,Z -48.355,A -90.000,B 90.000,C 0.000} C_DIS
LIN {X 94.048,Y -33.308,Z -47.934,A -90.000,B 90.000,C 0.000} C_DIS
LIN {X 94.008,Y -33.308,Z -47.725,A -90.000,B 90.000,C 0.000} C_DIS
LIN {X 93.969,Y -33.308,Z -47.446,A -90.000,B 90.000,C 0.000} C_DIS
LIN {X 93.970,Y -33.308,Z -47.410,A -90.000,B 90.000,C 0.000} C_DIS
LIN {X 93.976,Y -33.308,Z -46.998,A -90.000,B 90.000,C 0.000} C_DIS
LIN {X 94.004,Y -33.308,Z -46.687,A -90.000,B 90.000,C 0.000} C_DIS
LIN {X 94.082,Y -33.308,Z -46.377,A -90.000,B 90.000,C 0.000} C_DIS
LIN {X 94.223,Y -33.308,Z -45.886,A -90.000,B 90.000,C 0.000} C_DIS
LIN {X 94.352,Y -33.308,Z -45.554,A -90.000,B 90.000,C 0.000} C_DIS
LIN {X 94.522,Y -33.308,Z -45.163,A -90.000,B 90.000,C 0.000} C_DIS
LIN {X 94.682,Y -33.308,Z -44.819,A -90.000,B 90.000,C 0.000} C_DIS
LIN {X 94.808,Y -33.308,Z -44.577,A -90.000,B 90.000,C 0.000} C_DIS
LIN {X 94.938,Y -33.308,Z -44.340,A -90.000,B 90.000,C 0.000} C_DIS
LIN {X 95.287,Y -33.308,Z -43.751,A -90.000,B 90.000,C 0.000} C_DIS
LIN {X 95.352,Y -33.308,Z -43.638,A -90.000,B 90.000,C 0.000} C_DIS
LIN {X 95.579,Y -33.308,Z -43.305,A -90.000,B 90.000,C 0.000} C_DIS
LIN {X 96.023,Y -33.308,Z -42.688,A -90.000,B 90.000,C 0.000} C_DIS
LIN {X 96.804,Y -33.308,Z -41.778,A -90.000,B 90.000,C 0.000} C_DIS
LIN {X 97.620,Y -33.308,Z -40.978,A -90.000,B 90.000,C 0.000} C_DIS
LIN {X 98.293,Y -33.308,Z -40.401,A -90.000,B 90.000,C 0.000} C_DIS
LIN {X 98.488,Y -33.308,Z -40.239,A -90.000,B 90.000,C 0.000} C_DIS
LIN {X 99.372,Y -33.308,Z -39.589,A -90.000,B 90.000,C 0.000} C_DIS
LIN {X 100.004,Y -33.308,Z -39.176,A -90.000,B 90.000,C 0.000} C_DIS
LIN {X 100.704,Y -33.308,Z -38.748,A -90.000,B 90.000,C 0.000} C_DIS
LIN {X 101.666,Y -33.308,Z -38.226,A -90.000,B 90.000,C 0.000} C_DIS
LIN {X 102.746,Y -33.308,Z -37.714,A -90.000,B 90.000,C 0.000} C_DIS
LIN {X 103.228,Y -33.308,Z -37.494,A -90.000,B 90.000,C 0.000} C_DIS
LIN {X 104.493,Y -33.308,Z -36.935,A -90.000,B 90.000,C 0.000} C_DIS
LIN {X 105.393,Y -33.308,Z -36.556,A -90.000,B 90.000,C 0.000} C_DIS
LIN {X 106.867,Y -33.308,Z -35.970,A -90.000,B 90.000,C 0.000} C_DIS
LIN {X 107.391,Y -33.308,Z -35.771,A -90.000,B 90.000,C 0.000} C_DIS
LIN {X 107.871,Y -33.308,Z -35.598,A -90.000,B 90.000,C 0.000} C_DIS
LIN {X 108.337,Y -33.308,Z -35.443,A -90.000,B 90.000,C 0.000} C_DIS
LIN {X 108.769,Y -33.308,Z -35.328,A -90.000,B 90.000,C 0.000} C_DIS
LIN {X 109.226,Y -33.308,Z -35.225,A -90.000,B 90.000,C 0.000} C_DIS
LIN {X 109.649,Y -33.308,Z -35.169,A -90.000,B 90.000,C 0.000} C_DIS
LIN {X 110.108,Y -33.308,Z -35.113,A -90.000,B 90.000,C 0.000} C_DIS
LIN {X 110.614,Y -33.308,Z -35.106,A -90.000,B 90.000,C 0.000} C_DIS
LIN {X 110.969,Y -33.308,Z -35.118,A -90.000,B 90.000,C 0.000} C_DIS
LIN {X 111.443,Y -33.308,Z -35.160,A -90.000,B 90.000,C 0.000} C_DIS
LIN {X 112.073,Y -33.308,Z -35.278,A -90.000,B 90.000,C 0.000} C_DIS
LIN {X 112.435,Y -33.308,Z -35.371,A -90.000,B 90.000,C 0.000} C_DIS
LIN {X 112.884,Y -33.308,Z -35.505,A -90.000,B 90.000,C 0.000} C_DIS
LIN {X 113.055,Y -33.308,Z -35.560,A -90.000,B 90.000,C 0.000} C_DIS
LIN {X 113.513,Y -33.308,Z -35.750,A -90.000,B 90.000,C 0.000} C_DIS
LIN {X 113.987,Y -33.308,Z -35.977,A -90.000,B 90.000,C 0.000} C_DIS
LIN {X 114.418,Y -33.308,Z -36.210,A -90.000,B 90.000,C 0.000} C_DIS
LIN {X 114.548,Y -33.308,Z -36.291,A -90.000,B 90.000,C 0.000} C_DIS
LIN {X 114.952,Y -33.308,Z -36.567,A -90.000,B 90.000,C 0.000} C_DIS
LIN {X 115.073,Y -33.308,Z -36.664,A -90.000,B 90.000,C 0.000} C_DIS
LIN {X 115.430,Y -33.308,Z -36.965,A -90.000,B 90.000,C 0.000} C_DIS
LIN {X 115.520,Y -33.308,Z -37.046,A -90.000,B 90.000,C 0.000} C_DIS
LIN {X 115.872,Y -33.308,Z -37.410,A -90.000,B 90.000,C 0.000} C_DIS
LIN {X 116.081,Y -33.308,Z -37.633,A -90.000,B 90.000,C 0.000} C_DIS
LIN {X 116.439,Y -33.308,Z -38.088,A -90.000,B 90.000,C 0.000} C_DIS
LIN {X 116.700,Y -33.308,Z -38.500,A -90.000,B 90.000,C 0.000} C_DIS
LIN {X 116.930,Y -33.308,Z -38.965,A -90.000,B 90.000,C 0.000} C_DIS
LIN {X 117.059,Y -33.308,Z -39.250,A -90.000,B 90.000,C 0.000} C_DIS
LIN {X 117.105,Y -33.308,Z -39.367,A -90.000,B 90.000,C 0.000} C_DIS
LIN {X 117.260,Y -33.308,Z -39.781,A -90.000,B 90.000,C 0.000} C_DIS
LIN {X 117.391,Y -33.308,Z -40.285,A -90.000,B 90.000,C 0.000} C_DIS
LIN {X 117.462,Y -33.308,Z -40.593,A -90.000,B 90.000,C 0.000} C_DIS
LIN {X 117.541,Y -33.308,Z -41.113,A -90.000,B 90.000,C 0.000} C_DIS
LIN {X 117.596,Y -33.308,Z -41.528,A -90.000,B 90.000,C 0.000} C_DIS
LIN {X 117.631,Y -33.308,Z -41.885,A -90.000,B 90.000,C 0.000} C_DIS
LIN {X 117.656,Y -33.308,Z -42.390,A -90.000,B 90.000,C 0.000} C_DIS
LIN {X 117.668,Y -33.308,Z -42.698,A -90.000,B 90.000,C 0.000} C_DIS
LIN {X 117.664,Y -33.308,Z -42.870,A -90.000,B 90.000,C 0.000} C_DIS
LIN {X 117.651,Y -33.308,Z -43.202,A -90.000,B 90.000,C 0.000} C_DIS
LIN {X 117.607,Y -33.308,Z -43.724,A -90.000,B 90.000,C 0.000} C_DIS
LIN {X 117.565,Y -33.308,Z -44.127,A -90.000,B 90.000,C 0.000} C_DIS
LIN {X 117.487,Y -33.308,Z -44.644,A -90.000,B 90.000,C 0.000} C_DIS
LIN {X 117.396,Y -33.308,Z -45.126,A -90.000,B 90.000,C 0.000} C_DIS
LIN {X 117.258,Y -33.308,Z -45.748,A -90.000,B 90.000,C 0.000} C_DIS
LIN {X 117.117,Y -33.308,Z -46.220,A -90.000,B 90.000,C 0.000} C_DIS
LIN {X 116.895,Y -33.308,Z -46.951,A -90.000,B 90.000,C 0.000} C_DIS
LIN {X 116.548,Y -33.308,Z -47.851,A -90.000,B 90.000,C 0.000} C_DIS
LIN {X 116.366,Y -33.308,Z -48.292,A -90.000,B 90.000,C 0.000} C_DIS
LIN {X 115.865,Y -33.308,Z -49.367,A -90.000,B 90.000,C 0.000} C_DIS
LIN {X 115.244,Y -33.308,Z -50.609,A -90.000,B 90.000,C 0.000} C_DIS
LIN {X 114.588,Y -33.308,Z -51.909,A -90.000,B 90.000,C 0.000} C_DIS
LIN {X 113.934,Y -33.308,Z -53.246,A -90.000,B 90.000,C 0.000} C_DIS
LIN {X 113.270,Y -33.308,Z -54.704,A -90.000,B 90.000,C 0.000} C_DIS
LIN {X 112.799,Y -33.308,Z -55.830,A -90.000,B 90.000,C 0.000} C_DIS
LIN {X 112.208,Y -33.308,Z -57.403,A -90.000,B 90.000,C 0.000} C_DIS
LIN {X 111.674,Y -33.308,Z -59.009,A -90.000,B 90.000,C 0.000} C_DIS
LIN {X 111.248,Y -33.308,Z -60.488,A -90.000,B 90.000,C 0.000} C_DIS
LIN {X 110.729,Y -33.308,Z -62.393,A -90.000,B 90.000,C 0.000} C_DIS
LIN {X 110.160,Y -33.308,Z -64.412,A -90.000,B 90.000,C 0.000} C_DIS
LIN {X 110.004,Y -33.308,Z -64.935,A -90.000,B 90.000,C 0.000} C_DIS
LIN {X 109.346,Y -33.308,Z -66.982,A -90.000,B 90.000,C 0.000} C_DIS
LIN {X 109.232,Y -33.308,Z -67.288,A -90.000,B 90.000,C 0.000} C_DIS
LIN {X 108.444,Y -33.308,Z -69.382,A -90.000,B 90.000,C 0.000} C_DIS
LIN {X 108.266,Y -33.308,Z -69.835,A -90.000,B 90.000,C 0.000} C_DIS
LIN {X 107.794,Y -33.308,Z -70.994,A -90.000,B 90.000,C 0.000} C_DIS
LIN {X 107.256,Y -33.308,Z -72.303,A -90.000,B 90.000,C 0.000} C_DIS
LIN {X 106.195,Y -33.308,Z -74.712,A -90.000,B 90.000,C 0.000} C_DIS
LIN {X 106.111,Y -33.308,Z -74.887,A -90.000,B 90.000,C 0.000} C_DIS
LIN {X 105.114,Y -33.308,Z -76.881,A -90.000,B 90.000,C 0.000} C_DIS
LIN {X 104.890,Y -33.308,Z -77.312,A -90.000,B 90.000,C 0.000} C_DIS
LIN {X 103.836,Y -33.308,Z -79.207,A -90.000,B 90.000,C 0.000} C_DIS
LIN {X 102.834,Y -33.308,Z -80.849,A -90.000,B 90.000,C 0.000} C_DIS
LIN {X 101.634,Y -33.308,Z -82.673,A -90.000,B 90.000,C 0.000} C_DIS
LIN {X 101.240,Y -33.308,Z -83.244,A -90.000,B 90.000,C 0.000} C_DIS
LIN {X 99.546,Y -33.308,Z -85.657,A -90.000,B 90.000,C 0.000} C_DIS
LIN {X 98.229,Y -33.308,Z -87.504,A -90.000,B 90.000,C 0.000} C_DIS
LIN {X 98.180,Y -33.308,Z -87.629,A -90.000,B 90.000,C 0.000} C_DIS
LIN {X 98.064,Y -33.308,Z -88.111,A -90.000,B 90.000,C 0.000} C_DIS
LIN {X 97.969,Y -33.308,Z -88.865,A -90.000,B 90.000,C 0.000} C_DIS
LIN {X 97.901,Y -33.308,Z -89.382,A -90.000,B 90.000,C 0.000} C_DIS
LIN {X 97.865,Y -33.308,Z -89.837,A -90.000,B 90.000,C 0.000} C_DIS
LIN {X 97.733,Y -33.308,Z -91.279,A -90.000,B 90.000,C 0.000} C_DIS
LIN {X 97.623,Y -33.308,Z -92.457,A -90.000,B 90.000,C 0.000} C_DIS
LIN {X 97.552,Y -33.308,Z -93.287,A -90.000,B 90.000,C 0.000} C_DIS
LIN {X 97.509,Y -33.308,Z -93.694,A -90.000,B 90.000,C 0.000} C_DIS
LIN {X 97.414,Y -33.308,Z -94.676,A -90.000,B 90.000,C 0.000} C_DIS
LIN {X 97.372,Y -33.308,Z -94.986,A -90.000,B 90.000,C 0.000} C_DIS
LIN {X 97.285,Y -33.308,Z -95.433,A -90.000,B 90.000,C 0.000} C_DIS
LIN {X 97.119,Y -33.308,Z -96.227,A -90.000,B 90.000,C 0.000} C_DIS
LIN {X 97.045,Y -33.308,Z -96.601,A -90.000,B 90.000,C 0.000} C_DIS
LIN {X 96.908,Y -33.308,Z -97.043,A -90.000,B 90.000,C 0.000} C_DIS
LIN {X 96.769,Y -33.308,Z -97.537,A -90.000,B 90.000,C 0.000} C_DIS
LIN {X 96.634,Y -33.308,Z -97.977,A -90.000,B 90.000,C 0.000} C_DIS
LIN {X 96.334,Y -33.308,Z -98.850,A -90.000,B 90.000,C 0.000} C_DIS
LIN {X 96.013,Y -33.308,Z -99.690,A -90.000,B 90.000,C 0.000} C_DIS
LIN {X 95.928,Y -33.308,Z -99.925,A -90.000,B 90.000,C 0.000} C_DIS
LIN {X 95.649,Y -33.308,Z -100.828,A -90.000,B 90.000,C 0.000} C_DIS
LIN {X 95.323,Y -33.308,Z -102.043,A -90.000,B 90.000,C 0.000} C_DIS
LIN {X 95.241,Y -33.308,Z -102.351,A -90.000,B 90.000,C 0.000} C_DIS
LIN {X 95.051,Y -33.308,Z -103.217,A -90.000,B 90.000,C 0.000} C_DIS
LIN {X 94.944,Y -33.308,Z -103.628,A -90.000,B 90.000,C 0.000} C_DIS
LIN {X 94.789,Y -33.308,Z -104.484,A -90.000,B 90.000,C 0.000} C_DIS
LIN {X 94.769,Y -33.308,Z -105.092,A -90.000,B 90.000,C 0.000} C_DIS
LIN {X 94.825,Y -33.308,Z -105.535,A -90.000,B 90.000,C 0.000} C_DIS
LIN {X 94.856,Y -33.308,Z -105.851,A -90.000,B 90.000,C 0.000} C_DIS
LIN {X 95.002,Y -33.308,Z -106.701,A -90.000,B 90.000,C 0.000} C_DIS
LIN {X 95.038,Y -33.308,Z -106.942,A -90.000,B 90.000,C 0.000} C_DIS
LIN {X 95.205,Y -33.308,Z -108.222,A -90.000,B 90.000,C 0.000} C_DIS
LIN {X 95.230,Y -33.308,Z -108.662,A -90.000,B 90.000,C 0.000} C_DIS
LIN {X 95.307,Y -33.308,Z -110.265,A -90.000,B 90.000,C 0.000} C_DIS
LIN {X 95.323,Y -33.308,Z -112.125,A -90.000,B 90.000,C 0.000} C_DIS
LIN {X 95.307,Y -33.308,Z -114.151,A -90.000,B 90.000,C 0.000} C_DIS
LIN {X 95.302,Y -33.308,Z -116.279,A -90.000,B 90.000,C 0.000} C_DIS
LIN {X 95.323,Y -33.308,Z -117.389,A -90.000,B 90.000,C 0.000} C_DIS
LIN {X 95.334,Y -33.308,Z -118.447,A -90.000,B 90.000,C 0.000} C_DIS
LIN {X 95.376,Y -33.308,Z -120.630,A -90.000,B 90.000,C 0.000} C_DIS
LIN {X 95.400,Y -33.308,Z -122.474,A -90.000,B 90.000,C 0.000} C_DIS
LIN {X 95.406,Y -33.308,Z -122.794,A -90.000,B 90.000,C 0.000} C_DIS
LIN {X 95.393,Y -33.308,Z -124.484,A -90.000,B 90.000,C 0.000} C_DIS
LIN {X 95.391,Y -33.308,Z -125.017,A -90.000,B 90.000,C 0.000} C_DIS
LIN {X 95.301,Y -33.308,Z -127.090,A -90.000,B 90.000,C 0.000} C_DIS
LIN {X 95.147,Y -33.308,Z -129.239,A -90.000,B 90.000,C 0.000} C_DIS
LIN {X 95.032,Y -33.308,Z -130.547,A -90.000,B 90.000,C 0.000} C_DIS
LIN {X 94.906,Y -33.308,Z -132.014,A -90.000,B 90.000,C 0.000} C_DIS
LIN {X 94.794,Y -33.308,Z -133.244,A -90.000,B 90.000,C 0.000} C_DIS
LIN {X 94.690,Y -33.308,Z -134.437,A -90.000,B 90.000,C 0.000} C_DIS
LIN {X 94.574,Y -33.308,Z -135.866,A -90.000,B 90.000,C 0.000} C_DIS
LIN {X 94.441,Y -33.308,Z -137.453,A -90.000,B 90.000,C 0.000} C_DIS
LIN {X 94.261,Y -33.308,Z -139.565,A -90.000,B 90.000,C 0.000} C_DIS
LIN {X 94.103,Y -33.308,Z -141.377,A -90.000,B 90.000,C 0.000} C_DIS
LIN {X 93.737,Y -33.308,Z -145.077,A -90.000,B 90.000,C 0.000} C_DIS
LIN {X 93.286,Y -33.308,Z -148.833,A -90.000,B 90.000,C 0.000} C_DIS
LIN {X 92.728,Y -33.308,Z -152.506,A -90.000,B 90.000,C 0.000} C_DIS
LIN {X 92.062,Y -33.308,Z -156.124,A -90.000,B 90.000,C 0.000} C_DIS
LIN {X 91.977,Y -33.308,Z -156.539,A -90.000,B 90.000,C 0.000} C_DIS
LIN {X 91.202,Y -33.308,Z -160.130,A -90.000,B 90.000,C 0.000} C_DIS
LIN {X 90.319,Y -33.308,Z -163.722,A -90.000,B 90.000,C 0.000} C_DIS
LIN {X 89.777,Y -33.308,Z -165.683,A -90.000,B 90.000,C 0.000} C_DIS
LIN {X 89.325,Y -33.308,Z -167.341,A -90.000,B 90.000,C 0.000} C_DIS
LIN {X 88.717,Y -33.308,Z -169.382,A -90.000,B 90.000,C 0.000} C_DIS
LIN {X 88.270,Y -33.308,Z -170.910,A -90.000,B 90.000,C 0.000} C_DIS
LIN {X 87.624,Y -33.308,Z -172.978,A -90.000,B 90.000,C 0.000} C_DIS
LIN {X 87.203,Y -33.308,Z -174.351,A -90.000,B 90.000,C 0.000} C_DIS
LIN {X 86.469,Y -33.308,Z -176.652,A -90.000,B 90.000,C 0.000} C_DIS
LIN {X 86.153,Y -33.308,Z -177.653,A -90.000,B 90.000,C 0.000} C_DIS
LIN {X 85.207,Y -33.308,Z -180.630,A -90.000,B 90.000,C 0.000} C_DIS
LIN {X 84.884,Y -33.308,Z -181.640,A -90.000,B 90.000,C 0.000} C_DIS
LIN {X 84.327,Y -33.308,Z -183.396,A -90.000,B 90.000,C 0.000} C_DIS
LIN {X 84.001,Y -33.308,Z -184.412,A -90.000,B 90.000,C 0.000} C_DIS
LIN {X 83.495,Y -33.308,Z -186.005,A -90.000,B 90.000,C 0.000} C_DIS
LIN {X 82.332,Y -33.308,Z -189.646,A -90.000,B 90.000,C 0.000} C_DIS
LIN {X 81.876,Y -33.308,Z -191.061,A -90.000,B 90.000,C 0.000} C_DIS
LIN {X 81.486,Y -33.308,Z -192.261,A -90.000,B 90.000,C 0.000} C_DIS
LIN {X 80.883,Y -33.308,Z -194.073,A -90.000,B 90.000,C 0.000} C_DIS
LIN {X 80.403,Y -33.308,Z -195.495,A -90.000,B 90.000,C 0.000} C_DIS
LIN {X 79.963,Y -33.308,Z -196.764,A -90.000,B 90.000,C 0.000} C_DIS
LIN {X 79.272,Y -33.308,Z -198.723,A -90.000,B 90.000,C 0.000} C_DIS
LIN {X 78.668,Y -33.308,Z -200.383,A -90.000,B 90.000,C 0.000} C_DIS
LIN {X 77.882,Y -33.308,Z -202.522,A -90.000,B 90.000,C 0.000} C_DIS
LIN {X 77.206,Y -33.308,Z -204.307,A -90.000,B 90.000,C 0.000} C_DIS
LIN {X 76.223,Y -33.308,Z -206.885,A -90.000,B 90.000,C 0.000} C_DIS
LIN {X 75.677,Y -33.308,Z -208.274,A -90.000,B 90.000,C 0.000} C_DIS
LIN {X 74.247,Y -33.308,Z -211.888,A -90.000,B 90.000,C 0.000} C_DIS
LIN {X 74.017,Y -33.308,Z -212.464,A -90.000,B 90.000,C 0.000} C_DIS
LIN {X 73.777,Y -33.308,Z -213.052,A -90.000,B 90.000,C 0.000} C_DIS
LIN {X 73.262,Y -33.308,Z -214.416,A -90.000,B 90.000,C 0.000} C_DIS
LIN {X 71.687,Y -33.308,Z -218.308,A -90.000,B 90.000,C 0.000} C_DIS
LIN {X 70.300,Y -33.308,Z -221.583,A -90.000,B 90.000,C 0.000} C_DIS
LIN {X 69.660,Y -33.308,Z -223.224,A -90.000,B 90.000,C 0.000} C_DIS
LIN {X 69.543,Y -33.308,Z -223.516,A -90.000,B 90.000,C 0.000} C_DIS
LIN {X 68.578,Y -33.308,Z -225.742,A -90.000,B 90.000,C 0.000} C_DIS
LIN {X 67.474,Y -33.308,Z -228.502,A -90.000,B 90.000,C 0.000} C_DIS
LIN {X 66.725,Y -33.308,Z -230.220,A -90.000,B 90.000,C 0.000} C_DIS
LIN {X 65.197,Y -33.308,Z -234.009,A -90.000,B 90.000,C 0.000} C_DIS
LIN {X 64.673,Y -33.308,Z -235.225,A -90.000,B 90.000,C 0.000} C_DIS
LIN {X 64.577,Y -33.308,Z -235.463,A -90.000,B 90.000,C 0.000} C_DIS
LIN {X 63.711,Y -33.308,Z -237.881,A -90.000,B 90.000,C 0.000} C_DIS
LIN {X 63.154,Y -33.308,Z -239.595,A -90.000,B 90.000,C 0.000} C_DIS
LIN {X 61.823,Y -33.308,Z -243.561,A -90.000,B 90.000,C 0.000} C_DIS
LIN {X 61.823,Y -60.000,Z -243.561,A -90.000,B 90.000,C 0.000} C_DIS
LIN {X 109.977,Y -60.000,Z -65.020,A -90.000,B 90.000,C 0.000} C_DIS
LIN {X 109.977,Y -31.308,Z -65.020,A -90.000,B 90.000,C 0.000} C_DIS
LIN {X 109.345,Y -31.309,Z -67.050,A -90.000,B 90.000,C 0.000} C_DIS
LIN {X 108.519,Y -31.309,Z -69.358,A -90.000,B 90.000,C 0.000} C_DIS
LIN {X 107.589,Y -31.310,Z -71.699,A -90.000,B 90.000,C 0.000} C_DIS
LIN {X 107.406,Y -31.310,Z -72.144,A -90.000,B 90.000,C 0.000} C_DIS
LIN {X 106.414,Y -31.310,Z -74.420,A -90.000,B 90.000,C 0.000} C_DIS
LIN {X 105.797,Y -31.310,Z -75.709,A -90.000,B 90.000,C 0.000} C_DIS
LIN {X 105.390,Y -31.311,Z -76.551,A -90.000,B 90.000,C 0.000} C_DIS
LIN {X 104.136,Y -31.311,Z -78.889,A -90.000,B 90.000,C 0.000} C_DIS
LIN {X 103.987,Y -31.311,Z -79.149,A -90.000,B 90.000,C 0.000} C_DIS
LIN {X 103.058,Y -31.312,Z -80.726,A -90.000,B 90.000,C 0.000} C_DIS
LIN {X 102.201,Y -31.314,Z -82.073,A -90.000,B 90.000,C 0.000} C_DIS
LIN {X 100.778,Y -31.316,Z -84.205,A -90.000,B 90.000,C 0.000} C_DIS
LIN {X 100.238,Y -31.318,Z -85.013,A -90.000,B 90.000,C 0.000} C_DIS
LIN {X 99.000,Y -31.323,Z -86.844,A -90.000,B 90.000,C 0.000} C_DIS
LIN {X 98.967,Y -31.332,Z -86.995,A -90.000,B 90.000,C 0.000} C_DIS
LIN {X 98.920,Y -31.348,Z -87.216,A -90.000,B 90.000,C 0.000} C_DIS
LIN {X 98.887,Y -31.379,Z -87.488,A -90.000,B 90.000,C 0.000} C_DIS
LIN {X 98.858,Y -31.410,Z -87.708,A -90.000,B 90.000,C 0.000} C_DIS
LIN {X 98.836,Y -31.430,Z -87.834,A -90.000,B 90.000,C 0.000} C_DIS
LIN {X 98.783,Y -31.446,Z -88.242,A -90.000,B 90.000,C 0.000} C_DIS
LIN {X 98.757,Y -31.447,Z -88.458,A -90.000,B 90.000,C 0.000} C_DIS
LIN {X 98.687,Y -31.470,Z -89.447,A -90.000,B 90.000,C 0.000} C_DIS
LIN {X 98.626,Y -31.478,Z -90.386,A -90.000,B 90.000,C 0.000} C_DIS
LIN {X 98.593,Y -31.493,Z -91.094,A -90.000,B 90.000,C 0.000} C_DIS
LIN {X 98.517,Y -31.506,Z -92.193,A -90.000,B 90.000,C 0.000} C_DIS
LIN {X 98.438,Y -31.517,Z -93.363,A -90.000,B 90.000,C 0.000} C_DIS
LIN {X 98.393,Y -31.526,Z -93.982,A -90.000,B 90.000,C 0.000} C_DIS
LIN {X 98.386,Y -31.526,Z -94.052,A -90.000,B 90.000,C 0.000} C_DIS
LIN {X 98.309,Y -31.518,Z -94.678,A -90.000,B 90.000,C 0.000} C_DIS
LIN {X 98.296,Y -31.515,Z -94.762,A -90.000,B 90.000,C 0.000} C_DIS
LIN {X 98.240,Y -31.511,Z -95.104,A -90.000,B 90.000,C 0.000} C_DIS
LIN {X 98.153,Y -31.516,Z -95.617,A -90.000,B 90.000,C 0.000} C_DIS
LIN {X 98.147,Y -31.517,Z -95.656,A -90.000,B 90.000,C 0.000} C_DIS
LIN {X 98.040,Y -31.511,Z -96.107,A -90.000,B 90.000,C 0.000} C_DIS
LIN {X 97.908,Y -31.499,Z -96.636,A -90.000,B 90.000,C 0.000} C_DIS
LIN {X 97.856,Y -31.498,Z -96.853,A -90.000,B 90.000,C 0.000} C_DIS
LIN {X 97.795,Y -31.504,Z -97.093,A -90.000,B 90.000,C 0.000} C_DIS
LIN {X 97.731,Y -31.505,Z -97.310,A -90.000,B 90.000,C 0.000} C_DIS
LIN {X 97.691,Y -31.505,Z -97.451,A -90.000,B 90.000,C 0.000} C_DIS
LIN {X 97.534,Y -31.503,Z -97.973,A -90.000,B 90.000,C 0.000} C_DIS
LIN {X 97.512,Y -31.502,Z -98.037,A -90.000,B 90.000,C 0.000} C_DIS
LIN {X 97.449,Y -31.499,Z -98.225,A -90.000,B 90.000,C 0.000} C_DIS
LIN {X 97.220,Y -31.502,Z -98.911,A -90.000,B 90.000,C 0.000} C_DIS
LIN {X 97.129,Y -31.506,Z -99.199,A -90.000,B 90.000,C 0.000} C_DIS
LIN {X 96.856,Y -31.557,Z -100.197,A -90.000,B 90.000,C 0.000} C_DIS
LIN {X 96.788,Y -31.564,Z -100.457,A -90.000,B 90.000,C 0.000} C_DIS
LIN {X 96.645,Y -31.589,Z -101.066,A -90.000,B 90.000,C 0.000} C_DIS
LIN {X 96.467,Y -31.610,Z -101.852,A -90.000,B 90.000,C 0.000} C_DIS
LIN {X 96.413,Y -31.622,Z -102.130,A -90.000,B 90.000,C 0.000} C_DIS
LIN {X 96.319,Y -31.637,Z -102.572,A -90.000,B 90.000,C 0.000} C_DIS
LIN {X 96.163,Y -31.643,Z -103.313,A -90.000,B 90.000,C 0.000} C_DIS
LIN {X 96.146,Y -31.646,Z -103.419,A -90.000,B 90.000,C 0.000} C_DIS
LIN {X 96.065,Y -31.669,Z -103.863,A -90.000,B 90.000,C 0.000} C_DIS
LIN {X 95.977,Y -31.678,Z -104.421,A -90.000,B 90.000,C 0.000} C_DIS
LIN {X 95.966,Y -31.694,Z -104.606,A -90.000,B 90.000,C 0.000} C_DIS
LIN {X 95.955,Y -31.696,Z -105.036,A -90.000,B 90.000,C 0.000} C_DIS
LIN {X 95.957,Y -31.692,Z -105.100,A -90.000,B 90.000,C 0.000} C_DIS
LIN {X 95.993,Y -31.691,Z -105.411,A -90.000,B 90.000,C 0.000} C_DIS
LIN {X 96.023,Y -31.691,Z -105.700,A -90.000,B 90.000,C 0.000} C_DIS
LIN {X 96.046,Y -31.684,Z -105.891,A -90.000,B 90.000,C 0.000} C_DIS
LIN {X 96.135,Y -31.682,Z -106.424,A -90.000,B 90.000,C 0.000} C_DIS
LIN {X 96.180,Y -31.683,Z -106.702,A -90.000,B 90.000,C 0.000} C_DIS
LIN {X 96.218,Y -31.685,Z -106.962,A -90.000,B 90.000,C 0.000} C_DIS
LIN {X 96.361,Y -31.687,Z -108.023,A -90.000,B 90.000,C 0.000} C_DIS
LIN {X 96.382,Y -31.691,Z -108.199,A -90.000,B 90.000,C 0.000} C_DIS
LIN {X 96.451,Y -31.698,Z -109.374,A -90.000,B 90.000,C 0.000} C_DIS
LIN {X 96.496,Y -31.702,Z -110.180,A -90.000,B 90.000,C 0.000} C_DIS
LIN {X 96.511,Y -31.708,Z -110.861,A -90.000,B 90.000,C 0.000} C_DIS
LIN {X 96.527,Y -31.713,Z -111.973,A -90.000,B 90.000,C 0.000} C_DIS
LIN {X 96.527,Y -31.723,Z -114.154,A -90.000,B 90.000,C 0.000} C_DIS
LIN {X 96.532,Y -31.730,Z -116.088,A -90.000,B 90.000,C 0.000} C_DIS
LIN {X 96.534,Y -31.733,Z -116.288,A -90.000,B 90.000,C 0.000} C_DIS
LIN {X 96.556,Y -31.734,Z -117.375,A -90.000,B 90.000,C 0.000} C_DIS
LIN {X 96.571,Y -31.738,Z -118.274,A -90.000,B 90.000,C 0.000} C_DIS
LIN {X 96.620,Y -31.744,Z -120.484,A -90.000,B 90.000,C 0.000} C_DIS
LIN {X 96.650,Y -31.748,Z -122.414,A -90.000,B 90.000,C 0.000} C_DIS
LIN {X 96.656,Y -31.747,Z -122.768,A -90.000,B 90.000,C 0.000} C_DIS
LIN {X 96.650,Y -31.750,Z -124.038,A -90.000,B 90.000,C 0.000} C_DIS
LIN {X 96.648,Y -31.752,Z -124.862,A -90.000,B 90.000,C 0.000} C_DIS
LIN {X 96.646,Y -31.751,Z -125.021,A -90.000,B 90.000,C 0.000} C_DIS
LIN {X 96.597,Y -31.755,Z -126.285,A -90.000,B 90.000,C 0.000} C_DIS
LIN {X 96.564,Y -31.759,Z -127.146,A -90.000,B 90.000,C 0.000} C_DIS
LIN {X 96.529,Y -31.761,Z -127.679,A -90.000,B 90.000,C 0.000} C_DIS
LIN {X 96.421,Y -31.769,Z -129.330,A -90.000,B 90.000,C 0.000} C_DIS
LIN {X 96.357,Y -31.773,Z -130.105,A -90.000,B 90.000,C 0.000} C_DIS
LIN {X 96.225,Y -31.780,Z -131.731,A -90.000,B 90.000,C 0.000} C_DIS
LIN {X 95.994,Y -31.788,Z -134.442,A -90.000,B 90.000,C 0.000} C_DIS
LIN {X 95.922,Y -31.790,Z -135.346,A -90.000,B 90.000,C 0.000} C_DIS
LIN {X 95.703,Y -31.794,Z -138.031,A -90.000,B 90.000,C 0.000} C_DIS
LIN {X 95.409,Y -31.797,Z -141.481,A -90.000,B 90.000,C 0.000} C_DIS
LIN {X 95.290,Y -31.798,Z -142.699,A -90.000,B 90.000,C 0.000} C_DIS
LIN {X 95.047,Y -31.799,Z -145.165,A -90.000,B 90.000,C 0.000} C_DIS
LIN {X 94.900,Y -31.800,Z -146.411,A -90.000,B 90.000,C 0.000} C_DIS
LIN {X 94.602,Y -31.800,Z -148.897,A -90.000,B 90.000,C 0.000} C_DIS
LIN {X 94.589,Y -31.799,Z -148.990,A -90.000,B 90.000,C 0.000} C_DIS
LIN {X 94.419,Y -31.801,Z -150.127,A -90.000,B 90.000,C 0.000} C_DIS
LIN {X 94.053,Y -31.801,Z -152.539,A -90.000,B 90.000,C 0.000} C_DIS
LIN {X 94.025,Y -31.799,Z -152.703,A -90.000,B 90.000,C 0.000} C_DIS
LIN {X 93.837,Y -31.802,Z -153.750,A -90.000,B 90.000,C 0.000} C_DIS
LIN {X 93.399,Y -31.802,Z -156.129,A -90.000,B 90.000,C 0.000} C_DIS
LIN {X 93.361,Y -31.799,Z -156.322,A -90.000,B 90.000,C 0.000} C_DIS
LIN {X 93.315,Y -31.799,Z -156.544,A -90.000,B 90.000,C 0.000} C_DIS
LIN {X 93.067,Y -31.802,Z -157.727,A -90.000,B 90.000,C 0.000} C_DIS
LIN {X 92.552,Y -31.803,Z -160.117,A -90.000,B 90.000,C 0.000} C_DIS
LIN {X 92.486,Y -31.800,Z -160.406,A -90.000,B 90.000,C 0.000} C_DIS
LIN {X 92.282,Y -31.804,Z -161.261,A -90.000,B 90.000,C 0.000} C_DIS
LIN {X 91.681,Y -31.805,Z -163.709,A -90.000,B 90.000,C 0.000} C_DIS
LIN {X 91.598,Y -31.803,Z -164.037,A -90.000,B 90.000,C 0.000} C_DIS
LIN {X 91.396,Y -31.809,Z -164.795,A -90.000,B 90.000,C 0.000} C_DIS
LIN {X 91.208,Y -31.811,Z -165.481,A -90.000,B 90.000,C 0.000} C_DIS
LIN {X 90.604,Y -31.811,Z -167.690,A -90.000,B 90.000,C 0.000} C_DIS
LIN {X 90.422,Y -31.817,Z -168.325,A -90.000,B 90.000,C 0.000} C_DIS
LIN {X 90.000,Y -31.820,Z -169.757,A -90.000,B 90.000,C 0.000} C_DIS
LIN {X 89.553,Y -31.821,Z -171.285,A -90.000,B 90.000,C 0.000} C_DIS
LIN {X 89.399,Y -31.826,Z -171.796,A -90.000,B 90.000,C 0.000} C_DIS
LIN {X 88.911,Y -31.830,Z -173.373,A -90.000,B 90.000,C 0.000} C_DIS
LIN {X 88.551,Y -31.830,Z -174.548,A -90.000,B 90.000,C 0.000} C_DIS
LIN {X 88.365,Y -31.834,Z -175.154,A -90.000,B 90.000,C 0.000} C_DIS
LIN {X 88.088,Y -31.837,Z -176.031,A -90.000,B 90.000,C 0.000} C_DIS
LIN {X 87.537,Y -31.838,Z -177.772,A -90.000,B 90.000,C 0.000} C_DIS
LIN {X 86.964,Y -31.838,Z -179.579,A -90.000,B 90.000,C 0.000} C_DIS
LIN {X 86.596,Y -31.847,Z -180.764,A -90.000,B 90.000,C 0.000} C_DIS
LIN {X 86.083,Y -31.848,Z -182.378,A -90.000,B 90.000,C 0.000} C_DIS
LIN {X 85.728,Y -31.856,Z -183.525,A -90.000,B 90.000,C 0.000} C_DIS
LIN {X 85.308,Y -31.858,Z -184.844,A -90.000,B 90.000,C 0.000} C_DIS
LIN {X 84.888,Y -31.868,Z -186.202,A -90.000,B 90.000,C 0.000} C_DIS
LIN {X 84.535,Y -31.869,Z -187.314,A -90.000,B 90.000,C 0.000} C_DIS
LIN {X 84.163,Y -31.882,Z -188.522,A -90.000,B 90.000,C 0.000} C_DIS
LIN {X 83.688,Y -31.905,Z -190.084,A -90.000,B 90.000,C 0.000} C_DIS
LIN {X 83.361,Y -31.909,Z -191.113,A -90.000,B 90.000,C 0.000} C_DIS
LIN {X 82.865,Y -31.934,Z -192.719,A -90.000,B 90.000,C 0.000} C_DIS
LIN {X 82.534,Y -31.940,Z -193.734,A -90.000,B 90.000,C 0.000} C_DIS
LIN {X 81.937,Y -31.969,Z -195.595,A -90.000,B 90.000,C 0.000} C_DIS
LIN {X 81.732,Y -31.979,Z -196.222,A -90.000,B 90.000,C 0.000} C_DIS
LIN {X 81.619,Y -31.981,Z -196.554,A -90.000,B 90.000,C 0.000} C_DIS
LIN {X 81.438,Y -31.988,Z -197.094,A -90.000,B 90.000,C 0.000} C_DIS
LIN {X 80.719,Y -32.025,Z -199.233,A -90.000,B 90.000,C 0.000} C_DIS
LIN {X 80.528,Y -32.038,Z -199.790,A -90.000,B 90.000,C 0.000} C_DIS
LIN {X 80.423,Y -32.047,Z -200.100,A -90.000,B 90.000,C 0.000} C_DIS
LIN {X 80.034,Y -32.079,Z -201.237,A -90.000,B 90.000,C 0.000} C_DIS
LIN {X 79.384,Y -32.109,Z -203.074,A -90.000,B 90.000,C 0.000} C_DIS
LIN {X 79.142,Y -32.123,Z -203.745,A -90.000,B 90.000,C 0.000} C_DIS
LIN {X 78.516,Y -32.176,Z -205.497,A -90.000,B 90.000,C 0.000} C_DIS
LIN {X 77.783,Y -32.208,Z -207.480,A -90.000,B 90.000,C 0.000} C_DIS
LIN {X 77.504,Y -32.223,Z -208.218,A -90.000,B 90.000,C 0.000} C_DIS
LIN {X 77.374,Y -32.233,Z -208.568,A -90.000,B 90.000,C 0.000} C_DIS
LIN {X 76.770,Y -32.282,Z -210.180,A -90.000,B 90.000,C 0.000} C_DIS
LIN {X 75.727,Y -32.326,Z -212.881,A -90.000,B 90.000,C 0.000} C_DIS
LIN {X 75.614,Y -32.334,Z -213.174,A -90.000,B 90.000,C 0.000} C_DIS
LIN {X 75.411,Y -32.350,Z -213.694,A -90.000,B 90.000,C 0.000} C_DIS
LIN {X 74.921,Y -32.377,Z -215.035,A -90.000,B 90.000,C 0.000} C_DIS
LIN {X 74.460,Y -32.412,Z -216.222,A -90.000,B 90.000,C 0.000} C_DIS
LIN {X 73.789,Y -32.436,Z -217.912,A -90.000,B 90.000,C 0.000} C_DIS
LIN {X 73.386,Y -32.446,Z -218.920,A -90.000,B 90.000,C 0.000} C_DIS
LIN {X 73.104,Y -32.456,Z -219.600,A -90.000,B 90.000,C 0.000} C_DIS
LIN {X 72.019,Y -32.535,Z -222.255,A -90.000,B 90.000,C 0.000} C_DIS
LIN {X 71.711,Y -32.553,Z -223.062,A -90.000,B 90.000,C 0.000} C_DIS
LIN {X 71.516,Y -32.557,Z -223.565,A -90.000,B 90.000,C 0.000} C_DIS
LIN {X 71.260,Y -32.560,Z -224.215,A -90.000,B 90.000,C 0.000} C_DIS
LIN {X 70.328,Y -32.622,Z -226.429,A -90.000,B 90.000,C 0.000} C_DIS
LIN {X 69.512,Y -32.666,Z -228.509,A -90.000,B 90.000,C 0.000} C_DIS
LIN {X 69.399,Y -32.668,Z -228.792,A -90.000,B 90.000,C 0.000} C_DIS
LIN {X 69.236,Y -32.675,Z -229.207,A -90.000,B 90.000,C 0.000} C_DIS
LIN {X 68.505,Y -32.720,Z -230.920,A -90.000,B 90.000,C 0.000} C_DIS
LIN {X 67.709,Y -32.758,Z -232.921,A -90.000,B 90.000,C 0.000} C_DIS
LIN {X 67.369,Y -32.785,Z -233.785,A -90.000,B 90.000,C 0.000} C_DIS
LIN {X 66.991,Y -32.804,Z -234.734,A -90.000,B 90.000,C 0.000} C_DIS
LIN {X 66.496,Y -32.833,Z -235.902,A -90.000,B 90.000,C 0.000} C_DIS
LIN {X 66.393,Y -32.838,Z -236.157,A -90.000,B 90.000,C 0.000} C_DIS
LIN {X 65.807,Y -32.859,Z -237.809,A -90.000,B 90.000,C 0.000} C_DIS
LIN {X 65.569,Y -32.872,Z -238.482,A -90.000,B 90.000,C 0.000} C_DIS
LIN {X 65.211,Y -32.886,Z -239.590,A -90.000,B 90.000,C 0.000} C_DIS
LIN {X 65.035,Y -32.889,Z -240.132,A -90.000,B 90.000,C 0.000} C_DIS
LIN {X 63.891,Y -32.915,Z -243.561,A -90.000,B 90.000,C 0.000} C_DIS
LIN {X 63.891,Y -60.000,Z -243.561,A -90.000,B 90.000,C 0.000} C_DIS
LIN {X 80.885,Y -60.000,Z -204.298,A -90.000,B 90.000,C 0.000} C_DIS
LIN {X 80.885,Y -31.308,Z -204.298,A -90.000,B 90.000,C 0.000} C_DIS
LIN {X 80.819,Y -31.318,Z -204.478,A -90.000,B 90.000,C 0.000} C_DIS
LIN {X 80.549,Y -31.354,Z -205.259,A -90.000,B 90.000,C 0.000} C_DIS
LIN {X 80.170,Y -31.405,Z -206.342,A -90.000,B 90.000,C 0.000} C_DIS
LIN {X 79.521,Y -31.465,Z -208.135,A -90.000,B 90.000,C 0.000} C_DIS
LIN {X 79.244,Y -31.499,Z -208.887,A -90.000,B 90.000,C 0.000} C_DIS
LIN {X 78.457,Y -31.599,Z -211.024,A -90.000,B 90.000,C 0.000} C_DIS
LIN {X 77.714,Y -31.662,Z -212.981,A -90.000,B 90.000,C 0.000} C_DIS
LIN {X 77.489,Y -31.688,Z -213.578,A -90.000,B 90.000,C 0.000} C_DIS
LIN {X 77.192,Y -31.723,Z -214.356,A -90.000,B 90.000,C 0.000} C_DIS
LIN {X 76.708,Y -31.774,Z -215.701,A -90.000,B 90.000,C 0.000} C_DIS
LIN {X 76.216,Y -31.830,Z -216.984,A -90.000,B 90.000,C 0.000} C_DIS
LIN {X 75.848,Y -31.859,Z -217.923,A -90.000,B 90.000,C 0.000} C_DIS
LIN {X 75.461,Y -31.885,Z -218.905,A -90.000,B 90.000,C 0.000} C_DIS
LIN {X 75.160,Y -31.918,Z -219.678,A -90.000,B 90.000,C 0.000} C_DIS
LIN {X 73.820,Y -32.068,Z -222.989,A -90.000,B 90.000,C 0.000} C_DIS
LIN {X 73.775,Y -32.073,Z -223.107,A -90.000,B 90.000,C 0.000} C_DIS
LIN {X 73.380,Y -32.094,Z -224.141,A -90.000,B 90.000,C 0.000} C_DIS
LIN {X 73.074,Y -32.122,Z -224.934,A -90.000,B 90.000,C 0.000} C_DIS
LIN {X 72.147,Y -32.215,Z -227.153,A -90.000,B 90.000,C 0.000} C_DIS
LIN {X 71.665,Y -32.260,Z -228.392,A -90.000,B 90.000,C 0.000} C_DIS
LIN {X 71.041,Y -32.308,Z -229.986,A -90.000,B 90.000,C 0.000} C_DIS
LIN {X 70.323,Y -32.369,Z -231.677,A -90.000,B 90.000,C 0.000} C_DIS
LIN {X 69.403,Y -32.442,Z -234.005,A -90.000,B 90.000,C 0.000} C_DIS
LIN {X 68.833,Y -32.475,Z -235.442,A -90.000,B 90.000,C 0.000} C_DIS
LIN {X 68.346,Y -32.508,Z -236.596,A -90.000,B 90.000,C 0.000} C_DIS
LIN {X 68.245,Y -32.514,Z -236.842,A -90.000,B 90.000,C 0.000} C_DIS
LIN {X 67.446,Y -32.549,Z -239.094,A -90.000,B 90.000,C 0.000} C_DIS
LIN {X 67.201,Y -32.559,Z -239.850,A -90.000,B 90.000,C 0.000} C_DIS
LIN {X 66.934,Y -32.560,Z -240.673,A -90.000,B 90.000,C 0.000} C_DIS
LIN {X 65.969,Y -32.570,Z -243.561,A -90.000,B 90.000,C 0.000} C_DIS
LIN {X 65.969,Y -60.000,Z -243.561,A -90.000,B 90.000,C 0.000} C_DIS
LIN {X 77.916,Y -60.000,Z -217.932,A -90.000,B 90.000,C 0.000} C_DIS
LIN {X 77.916,Y -31.308,Z -217.932,A -90.000,B 90.000,C 0.000} C_DIS
LIN {X 77.211,Y -31.386,Z -219.746,A -90.000,B 90.000,C 0.000} C_DIS
LIN {X 76.958,Y -31.422,Z -220.400,A -90.000,B 90.000,C 0.000} C_DIS
LIN {X 75.770,Y -31.597,Z -223.361,A -90.000,B 90.000,C 0.000} C_DIS
LIN {X 75.627,Y -31.612,Z -223.713,A -90.000,B 90.000,C 0.000} C_DIS
LIN {X 75.249,Y -31.645,Z -224.712,A -90.000,B 90.000,C 0.000} C_DIS
LIN {X 75.054,Y -31.663,Z -225.221,A -90.000,B 90.000,C 0.000} C_DIS
LIN {X 74.889,Y -31.683,Z -225.650,A -90.000,B 90.000,C 0.000} C_DIS
LIN {X 73.967,Y -31.804,Z -227.877,A -90.000,B 90.000,C 0.000} C_DIS
LIN {X 73.642,Y -31.844,Z -228.714,A -90.000,B 90.000,C 0.000} C_DIS
LIN {X 72.861,Y -31.904,Z -230.710,A -90.000,B 90.000,C 0.000} C_DIS
LIN {X 72.143,Y -31.980,Z -232.410,A -90.000,B 90.000,C 0.000} C_DIS
LIN {X 71.405,Y -32.054,Z -234.284,A -90.000,B 90.000,C 0.000} C_DIS
LIN {X 71.104,Y -32.071,Z -235.043,A -90.000,B 90.000,C 0.000} C_DIS
LIN {X 70.652,Y -32.100,Z -236.182,A -90.000,B 90.000,C 0.000} C_DIS
LIN {X 70.163,Y -32.137,Z -237.344,A -90.000,B 90.000,C 0.000} C_DIS
LIN {X 70.079,Y -32.143,Z -237.550,A -90.000,B 90.000,C 0.000} C_DIS
LIN {X 69.307,Y -32.187,Z -239.731,A -90.000,B 90.000,C 0.000} C_DIS
LIN {X 69.176,Y -32.193,Z -240.136,A -90.000,B 90.000,C 0.000} C_DIS
LIN {X 68.804,Y -32.194,Z -241.281,A -90.000,B 90.000,C 0.000} C_DIS
LIN {X 68.041,Y -32.199,Z -243.561,A -90.000,B 90.000,C 0.000} C_DIS
LIN {X 68.041,Y -60.000,Z -243.561,A -90.000,B 90.000,C 0.000} C_DIS
LIN {X 75.634,Y -60.000,Z -228.924,A -90.000,B 90.000,C 0.000} C_DIS
LIN {X 75.634,Y -31.308,Z -228.924,A -90.000,B 90.000,C 0.000} C_DIS
LIN {X 75.555,Y -31.321,Z -229.131,A -90.000,B 90.000,C 0.000} C_DIS
LIN {X 74.638,Y -31.409,Z -231.483,A -90.000,B 90.000,C 0.000} C_DIS
LIN {X 73.932,Y -31.490,Z -233.160,A -90.000,B 90.000,C 0.000} C_DIS
LIN {X 73.776,Y -31.505,Z -233.556,A -90.000,B 90.000,C 0.000} C_DIS
LIN {X 73.323,Y -31.560,Z -234.711,A -90.000,B 90.000,C 0.000} C_DIS
LIN {X 72.423,Y -31.615,Z -236.976,A -90.000,B 90.000,C 0.000} C_DIS
LIN {X 71.907,Y -31.653,Z -238.204,A -90.000,B 90.000,C 0.000} C_DIS
LIN {X 71.871,Y -31.655,Z -238.299,A -90.000,B 90.000,C 0.000} C_DIS
LIN {X 71.573,Y -31.665,Z -239.135,A -90.000,B 90.000,C 0.000} C_DIS
LIN {X 71.139,Y -31.687,Z -240.360,A -90.000,B 90.000,C 0.000} C_DIS
LIN {X 71.050,Y -31.689,Z -240.631,A -90.000,B 90.000,C 0.000} C_DIS
LIN {X 70.635,Y -31.673,Z -241.895,A -90.000,B 90.000,C 0.000} C_DIS
LIN {X 70.071,Y -31.656,Z -243.561,A -90.000,B 90.000,C 0.000} C_DIS
LIN {X 70.071,Y -60.000,Z -243.561,A -90.000,B 90.000,C 0.000} C_DIS
LIN {X -98.559,Y -60.000,Z -243.561,A -90.000,B 90.000,C 0.000} C_DIS
LIN {X -98.559,Y -32.219,Z -243.561,A -90.000,B 90.000,C 0.000} C_DIS
LIN {X -98.554,Y -32.212,Z -243.551,A -90.000,B 90.000,C 0.000} C_DIS
LIN {X -98.499,Y -32.139,Z -243.439,A -90.000,B 90.000,C 0.000} C_DIS
LIN {X -98.460,Y -32.095,Z -243.370,A -90.000,B 90.000,C 0.000} C_DIS
LIN {X -98.323,Y -31.981,Z -243.162,A -90.000,B 90.000,C 0.000} C_DIS
LIN {X -98.100,Y -31.868,Z -242.897,A -90.000,B 90.000,C 0.000} C_DIS
LIN {X -97.628,Y -31.791,Z -242.494,A -90.000,B 90.000,C 0.000} C_DIS
LIN {X -95.558,Y -31.785,Z -241.054,A -90.000,B 90.000,C 0.000} C_DIS
LIN {X -92.950,Y -31.795,Z -239.216,A -90.000,B 90.000,C 0.000} C_DIS
LIN {X -91.063,Y -31.798,Z -237.883,A -90.000,B 90.000,C 0.000} C_DIS
LIN {X -90.878,Y -31.795,Z -237.760,A -90.000,B 90.000,C 0.000} C_DIS
LIN {X -90.416,Y -31.789,Z -237.453,A -90.000,B 90.000,C 0.000} C_DIS
LIN {X -89.171,Y -31.789,Z -236.642,A -90.000,B 90.000,C 0.000} C_DIS
LIN {X -86.637,Y -31.805,Z -234.972,A -90.000,B 90.000,C 0.000} C_DIS
LIN {X -82.957,Y -31.818,Z -232.536,A -90.000,B 90.000,C 0.000} C_DIS
LIN {X -82.318,Y -31.807,Z -232.133,A -90.000,B 90.000,C 0.000} C_DIS
LIN {X -81.570,Y -31.812,Z -231.672,A -90.000,B 90.000,C 0.000} C_DIS
LIN {X -80.084,Y -31.818,Z -230.766,A -90.000,B 90.000,C 0.000} C_DIS
LIN {X -74.585,Y -31.830,Z -227.405,A -90.000,B 90.000,C 0.000} C_DIS
LIN {X -73.868,Y -31.815,Z -226.988,A -90.000,B 90.000,C 0.000} C_DIS
LIN {X -73.512,Y -31.815,Z -226.790,A -90.000,B 90.000,C 0.000} C_DIS
LIN {X -67.471,Y -31.829,Z -223.435,A -90.000,B 90.000,C 0.000} C_DIS
LIN {X -65.890,Y -31.842,Z -222.568,A -90.000,B 90.000,C 0.000} C_DIS
LIN {X -65.279,Y -31.842,Z -222.241,A -90.000,B 90.000,C 0.000} C_DIS
LIN {X -64.895,Y -31.843,Z -222.040,A -90.000,B 90.000,C 0.000} C_DIS
LIN {X -61.202,Y -31.877,Z -220.127,A -90.000,B 90.000,C 0.000} C_DIS
LIN {X -56.966,Y -31.910,Z -217.943,A -90.000,B 90.000,C 0.000} C_DIS
LIN {X -56.376,Y -31.911,Z -217.643,A -90.000,B 90.000,C 0.000} C_DIS
LIN {X -55.251,Y -31.919,Z -217.077,A -90.000,B 90.000,C 0.000} C_DIS
LIN {X -51.125,Y -31.939,Z -215.009,A -90.000,B 90.000,C 0.000} C_DIS
LIN {X -48.459,Y -31.949,Z -213.684,A -90.000,B 90.000,C 0.000} C_DIS
LIN {X -45.957,Y -31.951,Z -212.429,A -90.000,B 90.000,C 0.000} C_DIS
LIN {X -44.997,Y -31.949,Z -211.950,A -90.000,B 90.000,C 0.000} C_DIS
LIN {X -42.110,Y -31.952,Z -210.522,A -90.000,B 90.000,C 0.000} C_DIS
LIN {X -41.672,Y -31.958,Z -210.300,A -90.000,B 90.000,C 0.000} C_DIS
LIN {X -38.518,Y -31.960,Z -208.655,A -90.000,B 90.000,C 0.000} C_DIS
LIN {X -37.474,Y -31.966,Z -208.106,A -90.000,B 90.000,C 0.000} C_DIS
LIN {X -36.583,Y -31.965,Z -207.631,A -90.000,B 90.000,C 0.000} C_DIS
LIN {X -36.086,Y -31.971,Z -207.360,A -90.000,B 90.000,C 0.000} C_DIS
LIN {X -34.332,Y -31.971,Z -206.379,A -90.000,B 90.000,C 0.000} C_DIS
LIN {X -34.079,Y -31.973,Z -206.236,A -90.000,B 90.000,C 0.000} C_DIS
LIN {X -31.797,Y -31.974,Z -204.935,A -90.000,B 90.000,C 0.000} C_DIS
LIN {X -31.327,Y -31.982,Z -204.660,A -90.000,B 90.000,C 0.000} C_DIS
LIN {X -30.894,Y -31.981,Z -204.397,A -90.000,B 90.000,C 0.000} C_DIS
LIN {X -30.255,Y -31.982,Z -204.008,A -90.000,B 90.000,C 0.000} C_DIS
LIN {X -27.732,Y -31.983,Z -202.453,A -90.000,B 90.000,C 0.000} C_DIS
LIN {X -27.300,Y -31.991,Z -202.179,A -90.000,B 90.000,C 0.000} C_DIS
LIN {X -26.939,Y -31.992,Z -201.941,A -90.000,B 90.000,C 0.000} C_DIS
LIN {X -24.350,Y -31.990,Z -200.216,A -90.000,B 90.000,C 0.000} C_DIS
LIN {X -23.890,Y -31.997,Z -199.902,A -90.000,B 90.000,C 0.000} C_DIS
LIN {X -21.009,Y -31.986,Z -197.863,A -90.000,B 90.000,C 0.000} C_DIS
LIN {X -20.645,Y -31.992,Z -197.597,A -90.000,B 90.000,C 0.000} C_DIS
LIN {X -17.653,Y -31.981,Z -195.341,A -90.000,B 90.000,C 0.000} C_DIS
LIN {X -17.282,Y -31.987,Z -195.053,A -90.000,B 90.000,C 0.000} C_DIS
LIN {X -14.284,Y -31.980,Z -192.660,A -90.000,B 90.000,C 0.000} C_DIS
LIN {X -13.919,Y -31.985,Z -192.362,A -90.000,B 90.000,C 0.000} C_DIS
LIN {X -10.796,Y -31.988,Z -189.753,A -90.000,B 90.000,C 0.000} C_DIS
LIN {X -10.424,Y -31.993,Z -189.437,A -90.000,B 90.000,C 0.000} C_DIS
LIN {X -7.959,Y -32.006,Z -187.308,A -90.000,B 90.000,C 0.000} C_DIS
LIN {X -7.232,Y -32.007,Z -186.683,A -90.000,B 90.000,C 0.000} C_DIS
LIN {X -6.721,Y -32.016,Z -186.234,A -90.000,B 90.000,C 0.000} C_DIS
LIN {X -4.759,Y -32.033,Z -184.480,A -90.000,B 90.000,C 0.000} C_DIS
LIN {X -3.698,Y -32.037,Z -183.536,A -90.000,B 90.000,C 0.000} C_DIS
LIN {X -3.072,Y -32.054,Z -182.969,A -90.000,B 90.000,C 0.000} C_DIS
LIN {X -0.503,Y -32.084,Z -180.574,A -90.000,B 90.000,C 0.000} C_DIS
LIN {X -0.178,Y -32.086,Z -180.278,A -90.000,B 90.000,C 0.000} C_DIS
LIN {X 0.290,Y -32.104,Z -179.837,A -90.000,B 90.000,C 0.000} C_DIS
LIN {X 2.732,Y -32.144,Z -177.430,A -90.000,B 90.000,C 0.000} C_DIS
LIN {X 3.031,Y -32.148,Z -177.145,A -90.000,B 90.000,C 0.000} C_DIS
LIN {X 3.412,Y -32.180,Z -176.757,A -90.000,B 90.000,C 0.000} C_DIS
LIN {X 3.456,Y -32.184,Z -176.712,A -90.000,B 90.000,C 0.000} C_DIS
LIN {X 3.548,Y -32.189,Z -176.610,A -90.000,B 90.000,C 0.000} C_DIS
LIN {X 4.398,Y -32.210,Z -175.690,A -90.000,B 90.000,C 0.000} C_DIS
LIN {X 5.593,Y -32.240,Z -174.396,A -90.000,B 90.000,C 0.000} C_DIS
LIN {X 5.864,Y -32.268,Z -174.083,A -90.000,B 90.000,C 0.000} C_DIS
LIN {X 6.137,Y -32.278,Z -173.714,A -90.000,B 90.000,C 0.000} C_DIS
LIN {X 6.344,Y -32.290,Z -173.448,A -90.000,B 90.000,C 0.000} C_DIS
LIN {X 7.223,Y -32.326,Z -172.334,A -90.000,B 90.000,C 0.000} C_DIS
LIN {X 7.700,Y -32.343,Z -171.733,A -90.000,B 90.000,C 0.000} C_DIS
LIN {X 7.754,Y -32.351,Z -171.661,A -90.000,B 90.000,C 0.000} C_DIS
LIN {X 8.258,Y -32.380,Z -170.804,A -90.000,B 90.000,C 0.000} C_DIS
LIN {X 8.737,Y -32.418,Z -169.981,A -90.000,B 90.000,C 0.000} C_DIS
LIN {X 8.893,Y -32.432,Z -169.722,A -90.000,B 90.000,C 0.000} C_DIS
LIN {X 9.019,Y -32.450,Z -169.507,A -90.000,B 90.000,C 0.000} C_DIS
LIN {X 9.151,Y -32.444,Z -169.110,A -90.000,B 90.000,C 0.000} C_DIS
LIN {X 9.388,Y -32.459,Z -168.359,A -90.000,B 90.000,C 0.000} C_DIS
LIN {X 9.750,Y -32.527,Z -167.146,A -90.000,B 90.000,C 0.000} C_DIS
LIN {X 9.770,Y -32.518,Z -166.897,A -90.000,B 90.000,C 0.000} C_DIS
LIN {X 9.801,Y -32.517,Z -166.392,A -90.000,B 90.000,C 0.000} C_DIS
LIN {X 9.771,Y -32.488,Z -165.777,A -90.000,B 90.000,C 0.000} C_DIS
LIN {X 9.761,Y -32.488,Z -165.574,A -90.000,B 90.000,C 0.000} C_DIS
LIN {X 9.742,Y -32.499,Z -165.275,A -90.000,B 90.000,C 0.000} C_DIS
LIN {X 9.554,Y -32.492,Z -164.026,A -90.000,B 90.000,C 0.000} C_DIS
LIN {X 9.226,Y -32.477,Z -162.845,A -90.000,B 90.000,C 0.000} C_DIS
LIN {X 9.105,Y -32.452,Z -162.575,A -90.000,B 90.000,C 0.000} C_DIS
LIN {X 8.658,Y -32.453,Z -161.673,A -90.000,B 90.000,C 0.000} C_DIS
LIN {X 8.545,Y -32.451,Z -161.454,A -90.000,B 90.000,C 0.000} C_DIS
LIN {X 8.510,Y -32.455,Z -161.392,A -90.000,B 90.000,C 0.000} C_DIS
LIN {X 8.046,Y -32.436,Z -160.822,A -90.000,B 90.000,C 0.000} C_DIS
LIN {X 7.636,Y -32.435,Z -160.329,A -90.000,B 90.000,C 0.000} C_DIS
LIN {X 7.574,Y -32.436,Z -160.251,A -90.000,B 90.000,C 0.000} C_DIS
LIN {X 7.437,Y -32.440,Z -160.071,A -90.000,B 90.000,C 0.000} C_DIS
LIN {X 7.064,Y -32.396,Z -159.758,A -90.000,B 90.000,C 0.000} C_DIS
LIN {X 5.919,Y -32.392,Z -158.877,A -90.000,B 90.000,C 0.000} C_DIS
LIN {X 5.899,Y -32.392,Z -158.862,A -90.000,B 90.000,C 0.000} C_DIS
LIN {X 5.188,Y -32.318,Z -158.478,A -90.000,B 90.000,C 0.000} C_DIS
LIN {X 4.786,Y -32.280,Z -158.253,A -90.000,B 90.000,C 0.000} C_DIS
LIN {X 3.893,Y -32.285,Z -157.811,A -90.000,B 90.000,C 0.000} C_DIS
LIN {X 3.153,Y -32.209,Z -157.547,A -90.000,B 90.000,C 0.000} C_DIS
LIN {X 2.417,Y -32.116,Z -157.266,A -90.000,B 90.000,C 0.000} C_DIS
LIN {X 1.775,Y -32.034,Z -157.013,A -90.000,B 90.000,C 0.000} C_DIS
LIN {X 0.806,Y -31.989,Z -156.692,A -90.000,B 90.000,C 0.000} C_DIS
LIN {X 0.375,Y -31.971,Z -156.546,A -90.000,B 90.000,C 0.000} C_DIS
LIN {X 0.332,Y -31.968,Z -156.529,A -90.000,B 90.000,C 0.000} C_DIS
LIN {X 0.022,Y -31.925,Z -156.435,A -90.000,B 90.000,C 0.000} C_DIS
LIN {X -0.083,Y -31.913,Z -156.399,A -90.000,B 90.000,C 0.000} C_DIS
LIN {X -0.482,Y -31.877,Z -156.250,A -90.000,B 90.000,C 0.000} C_DIS
LIN {X -1.756,Y -31.777,Z -155.754,A -90.000,B 90.000,C 0.000} C_DIS
LIN {X -1.872,Y -31.768,Z -155.707,A -90.000,B 90.000,C 0.000} C_DIS
LIN {X -2.698,Y -31.738,Z -155.422,A -90.000,B 90.000,C 0.000} C_DIS
LIN {X -2.842,Y -31.731,Z -155.369,A -90.000,B 90.000,C 0.000} C_DIS
LIN {X -3.095,Y -31.708,Z -155.283,A -90.000,B 90.000,C 0.000} C_DIS
LIN {X -3.800,Y -31.651,Z -155.040,A -90.000,B 90.000,C 0.000} C_DIS
LIN {X -4.259,Y -31.624,Z -154.873,A -90.000,B 90.000,C 0.000} C_DIS
LIN {X -4.384,Y -31.616,Z -154.823,A -90.000,B 90.000,C 0.000} C_DIS
LIN {X -5.131,Y -31.592,Z -154.508,A -90.000,B 90.000,C 0.000} C_DIS
LIN {X -5.200,Y -31.589,Z -154.476,A -90.000,B 90.000,C 0.000} C_DIS
LIN {X -6.122,Y -31.568,Z -154.101,A -90.000,B 90.000,C 0.000} C_DIS
LIN {X -6.411,Y -31.558,Z -153.986,A -90.000,B 90.000,C 0.000} C_DIS
LIN {X -6.599,Y -31.551,Z -153.908,A -90.000,B 90.000,C 0.000} C_DIS
LIN {X -7.964,Y -31.495,Z -153.334,A -90.000,B 90.000,C 0.000} C_DIS
LIN {X -8.399,Y -31.489,Z -153.145,A -90.000,B 90.000,C 0.000} C_DIS
LIN {X -8.475,Y -31.490,Z -153.114,A -90.000,B 90.000,C 0.000} C_DIS
LIN {X -9.387,Y -31.475,Z -152.668,A -90.000,B 90.000,C 0.000} C_DIS
LIN {X -9.850,Y -31.466,Z -152.438,A -90.000,B 90.000,C 0.000} C_DIS
LIN {X -11.571,Y -31.422,Z -151.585,A -90.000,B 90.000,C 0.000} C_DIS
LIN {X -11.713,Y -31.421,Z -151.521,A -90.000,B 90.000,C 0.000} C_DIS
LIN {X -11.800,Y -31.419,Z -151.479,A -90.000,B 90.000,C 0.000} C_DIS
LIN {X -12.153,Y -31.418,Z -151.304,A -90.000,B 90.000,C 0.000} C_DIS
LIN {X -12.424,Y -31.413,Z -151.147,A -90.000,B 90.000,C 0.000} C_DIS
LIN {X -14.401,Y -31.385,Z -150.001,A -90.000,B 90.000,C 0.000} C_DIS
LIN {X -15.350,Y -31.380,Z -149.484,A -90.000,B 90.000,C 0.000} C_DIS
LIN {X -15.836,Y -31.375,Z -149.209,A -90.000,B 90.000,C 0.000} C_DIS
LIN {X -16.614,Y -31.370,Z -148.684,A -90.000,B 90.000,C 0.000} C_DIS
LIN {X -18.809,Y -31.374,Z -147.274,A -90.000,B 90.000,C 0.000} C_DIS
LIN {X -19.408,Y -31.373,Z -146.889,A -90.000,B 90.000,C 0.000} C_DIS
LIN {X -19.757,Y -31.368,Z -146.640,A -90.000,B 90.000,C 0.000} C_DIS
LIN {X -19.859,Y -31.365,Z -146.564,A -90.000,B 90.000,C 0.000} C_DIS
LIN {X -20.117,Y -31.366,Z -146.370,A -90.000,B 90.000,C 0.000} C_DIS
LIN {X -20.996,Y -31.366,Z -145.696,A -90.000,B 90.000,C 0.000} C_DIS
LIN {X -22.101,Y -31.363,Z -144.851,A -90.000,B 90.000,C 0.000} C_DIS
LIN {X -23.320,Y -31.366,Z -143.952,A -90.000,B 90.000,C 0.000} C_DIS
LIN {X -23.522,Y -31.365,Z -143.789,A -90.000,B 90.000,C 0.000} C_DIS
LIN {X -23.832,Y -31.361,Z -143.520,A -90.000,B 90.000,C 0.000} C_DIS
LIN {X -25.390,Y -31.372,Z -142.159,A -90.000,B 90.000,C 0.000} C_DIS
LIN {X -25.642,Y -31.373,Z -141.935,A -90.000,B 90.000,C 0.000} C_DIS
LIN {X -26.277,Y -31.372,Z -141.367,A -90.000,B 90.000,C 0.000} C_DIS
LIN {X -26.679,Y -31.374,Z -141.018,A -90.000,B 90.000,C 0.000} C_DIS
LIN {X -27.074,Y -31.374,Z -140.669,A -90.000,B 90.000,C 0.000} C_DIS
LIN {X -27.158,Y -31.371,Z -140.582,A -90.000,B 90.000,C 0.000} C_DIS
LIN {X -27.519,Y -31.367,Z -140.204,A -90.000,B 90.000,C 0.000} C_DIS
LIN {X -28.121,Y -31.368,Z -139.572,A -90.000,B 90.000,C 0.000} C_DIS
LIN {X -28.206,Y -31.368,Z -139.486,A -90.000,B 90.000,C 0.000} C_DIS
LIN {X -30.088,Y -31.386,Z -137.561,A -90.000,B 90.000,C 0.000} C_DIS
LIN {X -30.453,Y -31.386,Z -137.165,A -90.000,B 90.000,C 0.000} C_DIS
LIN {X -30.508,Y -31.384,Z -137.096,A -90.000,B 90.000,C 0.000} C_DIS
LIN {X -30.737,Y -31.383,Z -136.802,A -90.000,B 90.000,C 0.000} C_DIS
LIN {X -32.037,Y -31.389,Z -135.126,A -90.000,B 90.000,C 0.000} C_DIS
LIN {X -33.003,Y -31.397,Z -133.903,A -90.000,B 90.000,C 0.000} C_DIS
LIN {X -33.181,Y -31.396,Z -133.664,A -90.000,B 90.000,C 0.000} C_DIS
LIN {X -33.290,Y -31.398,Z -133.516,A -90.000,B 90.000,C 0.000} C_DIS
LIN {X -33.466,Y -31.396,Z -133.239,A -90.000,B 90.000,C 0.000} C_DIS
LIN {X -35.106,Y -31.414,Z -130.658,A -90.000,B 90.000,C 0.000} C_DIS
LIN {X -35.352,Y -31.417,Z -130.266,A -90.000,B 90.000,C 0.000} C_DIS
LIN {X -35.497,Y -31.415,Z -130.021,A -90.000,B 90.000,C 0.000} C_DIS
LIN {X -35.571,Y -31.418,Z -129.895,A -90.000,B 90.000,C 0.000} C_DIS
LIN {X -35.595,Y -31.419,Z -129.848,A -90.000,B 90.000,C 0.000} C_DIS
LIN {X -37.254,Y -31.440,Z -126.481,A -90.000,B 90.000,C 0.000} C_DIS
LIN {X -37.333,Y -31.443,Z -126.307,A -90.000,B 90.000,C 0.000} C_DIS
LIN {X -37.407,Y -31.444,Z -126.119,A -90.000,B 90.000,C 0.000} C_DIS
LIN {X -37.716,Y -31.448,Z -125.305,A -90.000,B 90.000,C 0.000} C_DIS
LIN {X -38.462,Y -31.450,Z -123.292,A -90.000,B 90.000,C 0.000} C_DIS
LIN {X -38.605,Y -31.453,Z -122.903,A -90.000,B 90.000,C 0.000} C_DIS
LIN {X -38.713,Y -31.462,Z -122.606,A -90.000,B 90.000,C 0.000} C_DIS
LIN {X -38.839,Y -31.463,Z -122.147,A -90.000,B 90.000,C 0.000} C_DIS
LIN {X -39.301,Y -31.457,Z -120.379,A -90.000,B 90.000,C 0.000} C_DIS
LIN {X -39.477,Y -31.455,Z -119.714,A -90.000,B 90.000,C 0.000} C_DIS
LIN {X -39.611,Y -31.462,Z -119.207,A -90.000,B 90.000,C 0.000} C_DIS
LIN {X -39.732,Y -31.476,Z -118.734,A -90.000,B 90.000,C 0.000} C_DIS
LIN {X -39.821,Y -31.481,Z -118.314,A -90.000,B 90.000,C 0.000} C_DIS
LIN {X -39.850,Y -31.481,Z -118.150,A -90.000,B 90.000,C 0.000} C_DIS
LIN {X -40.262,Y -31.461,Z -115.712,A -90.000,B 90.000,C 0.000} C_DIS
LIN {X -40.295,Y -31.463,Z -115.510,A -90.000,B 90.000,C 0.000} C_DIS
LIN {X -40.429,Y -31.486,Z -114.674,A -90.000,B 90.000,C 0.000} C_DIS
LIN {X -40.484,Y -31.490,Z -114.214,A -90.000,B 90.000,C 0.000} C_DIS
LIN {X -40.551,Y -31.489,Z -113.416,A -90.000,B 90.000,C 0.000} C_DIS
LIN {X -40.669,Y -31.489,Z -112.160,A -90.000,B 90.000,C 0.000} C_DIS
LIN {X -40.717,Y -31.493,Z -111.639,A -90.000,B 90.000,C 0.000} C_DIS
LIN {X -40.741,Y -31.502,Z -111.353,A -90.000,B 90.000,C 0.000} C_DIS
LIN {X -40.808,Y -31.532,Z -110.608,A -90.000,B 90.000,C 0.000} C_DIS
LIN {X -40.813,Y -31.535,Z -110.529,A -90.000,B 90.000,C 0.000} C_DIS
LIN {X -40.880,Y -31.570,Z -109.897,A -90.000,B 90.000,C 0.000} C_DIS
LIN {X -40.955,Y -31.614,Z -109.515,A -90.000,B 90.000,C 0.000} C_DIS
LIN {X -40.976,Y -31.626,Z -109.374,A -90.000,B 90.000,C 0.000} C_DIS
LIN {X -41.069,Y -31.685,Z -109.036,A -90.000,B 90.000,C 0.000} C_DIS
LIN {X -41.094,Y -31.703,Z -108.923,A -90.000,B 90.000,C 0.000} C_DIS
LIN {X -41.194,Y -31.776,Z -108.453,A -90.000,B 90.000,C 0.000} C_DIS
LIN {X -41.226,Y -31.804,Z -108.335,A -90.000,B 90.000,C 0.000} C_DIS
LIN {X -41.232,Y -31.809,Z -108.312,A -90.000,B 90.000,C 0.000} C_DIS
LIN {X -41.322,Y -31.898,Z -107.911,A -90.000,B 90.000,C 0.000} C_DIS
LIN {X -41.345,Y -31.927,Z -107.793,A -90.000,B 90.000,C 0.000} C_DIS
LIN {X -41.472,Y -32.138,Z -106.994,A -90.000,B 90.000,C 0.000} C_DIS
LIN {X -41.494,Y -32.140,Z -106.951,A -90.000,B 90.000,C 0.000} C_DIS
LIN {X -41.625,Y -32.162,Z -106.720,A -90.000,B 90.000,C 0.000} C_DIS
LIN {X -41.899,Y -32.160,Z -106.340,A -90.000,B 90.000,C 0.000} C_DIS
LIN {X -42.345,Y -32.169,Z -105.674,A -90.000,B 90.000,C 0.000} C_DIS
LIN {X -42.632,Y -32.194,Z -105.269,A -90.000,B 90.000,C 0.000} C_DIS
LIN {X -43.017,Y -32.213,Z -104.750,A -90.000,B 90.000,C 0.000} C_DIS
LIN {X -43.339,Y -32.214,Z -104.346,A -90.000,B 90.000,C 0.000} C_DIS
LIN {X -43.414,Y -32.212,Z -104.250,A -90.000,B 90.000,C 0.000} C_DIS
LIN {X -43.884,Y -32.217,Z -103.666,A -90.000,B 90.000,C 0.000} C_DIS
LIN {X -43.978,Y -32.220,Z -103.544,A -90.000,B 90.000,C 0.000} C_DIS
LIN {X -44.180,Y -32.222,Z -103.273,A -90.000,B 90.000,C 0.000} C_DIS
LIN {X -44.875,Y -32.211,Z -102.383,A -90.000,B 90.000,C 0.000} C_DIS
LIN {X -45.052,Y -32.213,Z -102.143,A -90.000,B 90.000,C 0.000} C_DIS
LIN {X -45.769,Y -32.214,Z -101.159,A -90.000,B 90.000,C 0.000} C_DIS
LIN {X -46.267,Y -32.230,Z -100.439,A -90.000,B 90.000,C 0.000} C_DIS
LIN {X -47.163,Y -32.274,Z -99.156,A -90.000,B 90.000,C 0.000} C_DIS
LIN {X -47.609,Y -32.282,Z -98.503,A -90.000,B 90.000,C 0.000} C_DIS
LIN {X -47.857,Y -32.293,Z -98.129,A -90.000,B 90.000,C 0.000} C_DIS
LIN {X -48.185,Y -32.312,Z -97.622,A -90.000,B 90.000,C 0.000} C_DIS
LIN {X -49.013,Y -32.359,Z -96.319,A -90.000,B 90.000,C 0.000} C_DIS
LIN {X -49.210,Y -32.360,Z -95.999,A -90.000,B 90.000,C 0.000} C_DIS
LIN {X -49.458,Y -32.352,Z -95.579,A -90.000,B 90.000,C 0.000} C_DIS
LIN {X -49.573,Y -32.349,Z -95.379,A -90.000,B 90.000,C 0.000} C_DIS
LIN {X -49.708,Y -32.350,Z -95.129,A -90.000,B 90.000,C 0.000} C_DIS
LIN {X -49.793,Y -32.353,Z -94.966,A -90.000,B 90.000,C 0.000} C_DIS
LIN {X -49.833,Y -32.355,Z -94.884,A -90.000,B 90.000,C 0.000} C_DIS
LIN {X -50.972,Y -32.454,Z -92.448,A -90.000,B 90.000,C 0.000} C_DIS
LIN {X -51.243,Y -32.471,Z -91.860,A -90.000,B 90.000,C 0.000} C_DIS
LIN {X -51.397,Y -32.480,Z -91.522,A -90.000,B 90.000,C 0.000} C_DIS
LIN {X -51.565,Y -32.498,Z -91.117,A -90.000,B 90.000,C 0.000} C_DIS
LIN {X -51.598,Y -32.498,Z -91.036,A -90.000,B 90.000,C 0.000} C_DIS
LIN {X -51.795,Y -32.506,Z -90.488,A -90.000,B 90.000,C 0.000} C_DIS
LIN {X -51.880,Y -32.512,Z -90.238,A -90.000,B 90.000,C 0.000} C_DIS
LIN {X -52.340,Y -32.556,Z -88.807,A -90.000,B 90.000,C 0.000} C_DIS
LIN {X -52.519,Y -32.570,Z -88.267,A -90.000,B 90.000,C 0.000} C_DIS
LIN {X -52.648,Y -32.580,Z -87.867,A -90.000,B 90.000,C 0.000} C_DIS
LIN {X -52.841,Y -32.591,Z -87.255,A -90.000,B 90.000,C 0.000} C_DIS
LIN {X -52.923,Y -32.594,Z -86.983,A -90.000,B 90.000,C 0.000} C_DIS
LIN {X -53.546,Y -32.593,Z -84.740,A -90.000,B 90.000,C 0.000} C_DIS
LIN {X -53.571,Y -32.594,Z -84.638,A -90.000,B 90.000,C 0.000} C_DIS
LIN {X -54.060,Y -32.634,Z -82.466,A -90.000,B 90.000,C 0.000} C_DIS
LIN {X -54.093,Y -32.639,Z -82.305,A -90.000,B 90.000,C 0.000} C_DIS
LIN {X -54.336,Y -32.651,Z -81.001,A -90.000,B 90.000,C 0.000} C_DIS
LIN {X -54.419,Y -32.657,Z -80.560,A -90.000,B 90.000,C 0.000} C_DIS
LIN {X -54.450,Y -32.660,Z -80.389,A -90.000,B 90.000,C 0.000} C_DIS
LIN {X -54.486,Y -32.662,Z -80.134,A -90.000,B 90.000,C 0.000} C_DIS
LIN {X -54.520,Y -32.667,Z -79.814,A -90.000,B 90.000,C 0.000} C_DIS
LIN {X -54.595,Y -32.695,Z -79.120,A -90.000,B 90.000,C 0.000} C_DIS
LIN {X -54.628,Y -32.705,Z -78.832,A -90.000,B 90.000,C 0.000} C_DIS
LIN {X -54.689,Y -32.717,Z -78.304,A -90.000,B 90.000,C 0.000} C_DIS
LIN {X -54.702,Y -32.721,Z -78.129,A -90.000,B 90.000,C 0.000} C_DIS
LIN {X -54.718,Y -32.738,Z -77.686,A -90.000,B 90.000,C 0.000} C_DIS
LIN {X -54.743,Y -32.763,Z -76.890,A -90.000,B 90.000,C 0.000} C_DIS
LIN {X -54.750,Y -32.770,Z -76.666,A -90.000,B 90.000,C 0.000} C_DIS
LIN {X -54.752,Y -32.777,Z -76.346,A -90.000,B 90.000,C 0.000} C_DIS
LIN {X -54.761,Y -32.777,Z -76.251,A -90.000,B 90.000,C 0.000} C_DIS
LIN {X -54.767,Y -32.777,Z -76.136,A -90.000,B 90.000,C 0.000} C_DIS
LIN {X -54.775,Y -32.805,Z -75.082,A -90.000,B 90.000,C 0.000} C_DIS
LIN {X -54.775,Y -32.805,Z -74.830,A -90.000,B 90.000,C 0.000} C_DIS
LIN {X -54.789,Y -32.804,Z -74.612,A -90.000,B 90.000,C 0.000} C_DIS
LIN {X -54.794,Y -32.806,Z -74.468,A -90.000,B 90.000,C 0.000} C_DIS
LIN {X -54.786,Y -32.811,Z -74.296,A -90.000,B 90.000,C 0.000} C_DIS
LIN {X -54.735,Y -32.836,Z -73.586,A -90.000,B 90.000,C 0.000} C_DIS
LIN {X -54.725,Y -32.836,Z -73.452,A -90.000,B 90.000,C 0.000} C_DIS
LIN {X -54.714,Y -32.840,Z -73.306,A -90.000,B 90.000,C 0.000} C_DIS
LIN {X -54.720,Y -32.840,Z -72.990,A -90.000,B 90.000,C 0.000} C_DIS
LIN {X -54.719,Y -32.840,Z -72.864,A -90.000,B 90.000,C 0.000} C_DIS
LIN {X -54.692,Y -32.849,Z -72.505,A -90.000,B 90.000,C 0.000} C_DIS
LIN {X -54.676,Y -32.853,Z -72.383,A -90.000,B 90.000,C 0.000} C_DIS
LIN {X -54.639,Y -32.863,Z -72.153,A -90.000,B 90.000,C 0.000} C_DIS
LIN {X -54.548,Y -32.878,Z -71.603,A -90.000,B 90.000,C 0.000} C_DIS
LIN {X -54.535,Y -32.878,Z -71.329,A -90.000,B 90.000,C 0.000} C_DIS
LIN {X -54.513,Y -32.881,Z -71.070,A -90.000,B 90.000,C 0.000} C_DIS
LIN {X -54.475,Y -32.888,Z -70.824,A -90.000,B 90.000,C 0.000} C_DIS
LIN {X -54.468,Y -32.890,Z -70.796,A -90.000,B 90.000,C 0.000} C_DIS
LIN {X -54.420,Y -32.898,Z -70.611,A -90.000,B 90.000,C 0.000} C_DIS
LIN {X -54.243,Y -32.916,Z -69.968,A -90.000,B 90.000,C 0.000} C_DIS
LIN {X -54.197,Y -32.916,Z -69.640,A -90.000,B 90.000,C 0.000} C_DIS
LIN {X -54.181,Y -32.917,Z -69.541,A -90.000,B 90.000,C 0.000} C_DIS
LIN {X -54.171,Y -32.919,Z -69.490,A -90.000,B 90.000,C 0.000} C_DIS
LIN {X -54.130,Y -32.929,Z -69.325,A -90.000,B 90.000,C 0.000} C_DIS
LIN {X -54.060,Y -32.930,Z -69.092,A -90.000,B 90.000,C 0.000} C_DIS
LIN {X -53.931,Y -32.931,Z -68.775,A -90.000,B 90.000,C 0.000} C_DIS
LIN {X -53.659,Y -32.943,Z -68.246,A -90.000,B 90.000,C 0.000} C_DIS
LIN {X -53.567,Y -32.948,Z -68.065,A -90.000,B 90.000,C 0.000} C_DIS
LIN {X -53.546,Y -32.949,Z -68.008,A -90.000,B 90.000,C 0.000} C_DIS
LIN {X -53.501,Y -32.947,Z -67.887,A -90.000,B 90.000,C 0.000} C_DIS
LIN {X -53.486,Y -32.946,Z -67.845,A -90.000,B 90.000,C 0.000} C_DIS
LIN {X -53.457,Y -32.942,Z -67.772,A -90.000,B 90.000,C 0.000} C_DIS
LIN {X -53.421,Y -32.937,Z -67.691,A -90.000,B 90.000,C 0.000} C_DIS
LIN {X -53.361,Y -32.931,Z -67.573,A -90.000,B 90.000,C 0.000} C_DIS
LIN {X -53.172,Y -32.917,Z -67.233,A -90.000,B 90.000,C 0.000} C_DIS
LIN {X -53.083,Y -32.913,Z -67.098,A -90.000,B 90.000,C 0.000} C_DIS
LIN {X -53.028,Y -32.911,Z -67.024,A -90.000,B 90.000,C 0.000} C_DIS
LIN {X -52.958,Y -32.911,Z -66.938,A -90.000,B 90.000,C 0.000} C_DIS
LIN {X -52.788,Y -32.913,Z -66.743,A -90.000,B 90.000,C 0.000} C_DIS
LIN {X -52.465,Y -32.918,Z -66.403,A -90.000,B 90.000,C 0.000} C_DIS
LIN {X -52.329,Y -32.912,Z -66.263,A -90.000,B 90.000,C 0.000} C_DIS
LIN {X -51.959,Y -32.876,Z -65.887,A -90.000,B 90.000,C 0.000} C_DIS
LIN {X -51.629,Y -32.850,Z -65.550,A -90.000,B 90.000,C 0.000} C_DIS
LIN {X -51.556,Y -32.845,Z -65.482,A -90.000,B 90.000,C 0.000} C_DIS
LIN {X -51.455,Y -32.841,Z -65.398,A -90.000,B 90.000,C 0.000} C_DIS
LIN {X -51.172,Y -32.834,Z -65.188,A -90.000,B 90.000,C 0.000} C_DIS
LIN {X -51.051,Y -32.829,Z -65.113,A -90.000,B 90.000,C 0.000} C_DIS
LIN {X -51.003,Y -32.827,Z -65.080,A -90.000,B 90.000,C 0.000} C_DIS
LIN {X -50.576,Y -32.791,Z -64.795,A -90.000,B 90.000,C 0.000} C_DIS
LIN {X -50.105,Y -32.741,Z -64.486,A -90.000,B 90.000,C 0.000} C_DIS
LIN {X -50.019,Y -32.733,Z -64.432,A -90.000,B 90.000,C 0.000} C_DIS
LIN {X -49.660,Y -32.703,Z -64.224,A -90.000,B 90.000,C 0.000} C_DIS
LIN {X -49.507,Y -32.693,Z -64.135,A -90.000,B 90.000,C 0.000} C_DIS
LIN {X -49.401,Y -32.688,Z -64.078,A -90.000,B 90.000,C 0.000} C_DIS
LIN {X -48.827,Y -32.665,Z -63.791,A -90.000,B 90.000,C 0.000} C_DIS
LIN {X -48.626,Y -32.652,Z -63.696,A -90.000,B 90.000,C 0.000} C_DIS
LIN {X -48.478,Y -32.644,Z -63.640,A -90.000,B 90.000,C 0.000} C_DIS
LIN {X -47.250,Y -32.596,Z -63.215,A -90.000,B 90.000,C 0.000} C_DIS
LIN {X -46.099,Y -32.548,Z -62.809,A -90.000,B 90.000,C 0.000} C_DIS
LIN {X -45.949,Y -32.542,Z -62.761,A -90.000,B 90.000,C 0.000} C_DIS
LIN {X -45.678,Y -32.536,Z -62.683,A -90.000,B 90.000,C 0.000} C_DIS
LIN {X -45.226,Y -32.528,Z -62.561,A -90.000,B 90.000,C 0.000} C_DIS
LIN {X -45.026,Y -32.520,Z -62.509,A -90.000,B 90.000,C 0.000} C_DIS
LIN {X -44.357,Y -32.503,Z -62.356,A -90.000,B 90.000,C 0.000} C_DIS
LIN {X -44.014,Y -32.494,Z -62.278,A -90.000,B 90.000,C 0.000} C_DIS
LIN {X -43.437,Y -32.481,Z -62.150,A -90.000,B 90.000,C 0.000} C_DIS
LIN {X -43.082,Y -32.479,Z -62.084,A -90.000,B 90.000,C 0.000} C_DIS
LIN {X -42.020,Y -32.445,Z -61.897,A -90.000,B 90.000,C 0.000} C_DIS
LIN {X -41.135,Y -32.409,Z -61.747,A -90.000,B 90.000,C 0.000} C_DIS
LIN {X -40.213,Y -32.395,Z -61.642,A -90.000,B 90.000,C 0.000} C_DIS
LIN {X -40.015,Y -32.394,Z -61.626,A -90.000,B 90.000,C 0.000} C_DIS
LIN {X -39.731,Y -32.381,Z -61.614,A -90.000,B 90.000,C 0.000} C_DIS
LIN {X -39.340,Y -32.369,Z -61.609,A -90.000,B 90.000,C 0.000} C_DIS
LIN {X -39.194,Y -32.364,Z -61.605,A -90.000,B 90.000,C 0.000} C_DIS
LIN {X -36.959,Y -32.312,Z -61.526,A -90.000,B 90.000,C 0.000} C_DIS
LIN {X -36.813,Y -32.303,Z -61.523,A -90.000,B 90.000,C 0.000} C_DIS
LIN {X -36.693,Y -32.299,Z -61.525,A -90.000,B 90.000,C 0.000} C_DIS
LIN {X -35.809,Y -32.275,Z -61.559,A -90.000,B 90.000,C 0.000} C_DIS
LIN {X -35.597,Y -32.263,Z -61.573,A -90.000,B 90.000,C 0.000} C_DIS
LIN {X -35.246,Y -32.250,Z -61.608,A -90.000,B 90.000,C 0.000} C_DIS
LIN {X -33.333,Y -32.169,Z -61.827,A -90.000,B 90.000,C 0.000} C_DIS
LIN {X -33.094,Y -32.161,Z -61.857,A -90.000,B 90.000,C 0.000} C_DIS
LIN {X -32.842,Y -32.156,Z -61.897,A -90.000,B 90.000,C 0.000} C_DIS
LIN {X -32.241,Y -32.142,Z -62.002,A -90.000,B 90.000,C 0.000} C_DIS
LIN {X -30.710,Y -32.101,Z -62.281,A -90.000,B 90.000,C 0.000} C_DIS
LIN {X -30.473,Y -32.093,Z -62.326,A -90.000,B 90.000,C 0.000} C_DIS
LIN {X -30.038,Y -32.084,Z -62.417,A -90.000,B 90.000,C 0.000} C_DIS
LIN {X -28.535,Y -32.058,Z -62.750,A -90.000,B 90.000,C 0.000} C_DIS
LIN {X -27.792,Y -32.048,Z -62.918,A -90.000,B 90.000,C 0.000} C_DIS
LIN {X -27.653,Y -32.048,Z -62.952,A -90.000,B 90.000,C 0.000} C_DIS
LIN {X -27.475,Y -32.050,Z -62.997,A -90.000,B 90.000,C 0.000} C_DIS
LIN {X -26.818,Y -32.049,Z -63.175,A -90.000,B 90.000,C 0.000} C_DIS
LIN {X -25.508,Y -32.061,Z -63.518,A -90.000,B 90.000,C 0.000} C_DIS
LIN {X -25.425,Y -32.063,Z -63.541,A -90.000,B 90.000,C 0.000} C_DIS
LIN {X -24.069,Y -32.105,Z -63.953,A -90.000,B 90.000,C 0.000} C_DIS
LIN {X -23.712,Y -32.106,Z -64.067,A -90.000,B 90.000,C 0.000} C_DIS
LIN {X -23.604,Y -32.116,Z -64.094,A -90.000,B 90.000,C 0.000} C_DIS
LIN {X -23.321,Y -32.128,Z -64.178,A -90.000,B 90.000,C 0.000} C_DIS
LIN {X -22.701,Y -32.158,Z -64.372,A -90.000,B 90.000,C 0.000} C_DIS
LIN {X -22.633,Y -32.170,Z -64.387,A -90.000,B 90.000,C 0.000} C_DIS
LIN {X -22.521,Y -32.246,Z -64.373,A -90.000,B 90.000,C 0.000} C_DIS
LIN {X -22.493,Y -32.247,Z -64.290,A -90.000,B 90.000,C 0.000} C_DIS
LIN {X -22.255,Y -32.258,Z -63.612,A -90.000,B 90.000,C 0.000} C_DIS
LIN {X -22.222,Y -32.255,Z -63.534,A -90.000,B 90.000,C 0.000} C_DIS
LIN {X -22.124,Y -32.251,Z -63.313,A -90.000,B 90.000,C 0.000} C_DIS
LIN {X -22.055,Y -32.247,Z -63.162,A -90.000,B 90.000,C 0.000} C_DIS
LIN {X -22.011,Y -32.250,Z -63.073,A -90.000,B 90.000,C 0.000} C_DIS
LIN {X -21.845,Y -32.267,Z -62.759,A -90.000,B 90.000,C 0.000} C_DIS
LIN {X -21.733,Y -32.281,Z -62.561,A -90.000,B 90.000,C 0.000} C_DIS
LIN {X -21.560,Y -32.273,Z -62.272,A -90.000,B 90.000,C 0.000} C_DIS
LIN {X -21.509,Y -32.268,Z -62.188,A -90.000,B 90.000,C 0.000} C_DIS
LIN {X -21.427,Y -32.254,Z -62.063,A -90.000,B 90.000,C 0.000} C_DIS
LIN {X -21.340,Y -32.242,Z -61.940,A -90.000,B 90.000,C 0.000} C_DIS
LIN {X -21.080,Y -32.225,Z -61.616,A -90.000,B 90.000,C 0.000} C_DIS
LIN {X -21.000,Y -32.217,Z -61.527,A -90.000,B 90.000,C 0.000} C_DIS
LIN {X -20.923,Y -32.213,Z -61.449,A -90.000,B 90.000,C 0.000} C_DIS
LIN {X -20.625,Y -32.206,Z -61.163,A -90.000,B 90.000,C 0.000} C_DIS
LIN {X -20.551,Y -32.204,Z -61.098,A -90.000,B 90.000,C 0.000} C_DIS
LIN {X -20.488,Y -32.201,Z -61.048,A -90.000,B 90.000,C 0.000} C_DIS
LIN {X -20.225,Y -32.196,Z -60.857,A -90.000,B 90.000,C 0.000} C_DIS
LIN {X -20.165,Y -32.191,Z -60.817,A -90.000,B 90.000,C 0.000} C_DIS
LIN {X -19.749,Y -32.167,Z -60.549,A -90.000,B 90.000,C 0.000} C_DIS
LIN {X -19.656,Y -32.164,Z -60.493,A -90.000,B 90.000,C 0.000} C_DIS
LIN {X -19.416,Y -32.158,Z -60.354,A -90.000,B 90.000,C 0.000} C_DIS
LIN {X -19.280,Y -32.156,Z -60.279,A -90.000,B 90.000,C 0.000} C_DIS
LIN {X -19.155,Y -32.160,Z -60.219,A -90.000,B 90.000,C 0.000} C_DIS
LIN {X -18.914,Y -32.172,Z -60.113,A -90.000,B 90.000,C 0.000} C_DIS
LIN {X -18.480,Y -32.190,Z -59.929,A -90.000,B 90.000,C 0.000} C_DIS
LIN {X -18.180,Y -32.193,Z -59.818,A -90.000,B 90.000,C 0.000} C_DIS
LIN {X -17.710,Y -32.206,Z -59.657,A -90.000,B 90.000,C 0.000} C_DIS
LIN {X -17.505,Y -32.210,Z -59.589,A -90.000,B 90.000,C 0.000} C_DIS
LIN {X -17.369,Y -32.214,Z -59.547,A -90.000,B 90.000,C 0.000} C_DIS
LIN {X -17.177,Y -32.211,Z -59.494,A -90.000,B 90.000,C 0.000} C_DIS
LIN {X -16.984,Y -32.206,Z -59.443,A -90.000,B 90.000,C 0.000} C_DIS
LIN {X -16.489,Y -32.190,Z -59.316,A -90.000,B 90.000,C 0.000} C_DIS
LIN {X -16.306,Y -32.189,Z -59.275,A -90.000,B 90.000,C 0.000} C_DIS
LIN {X -16.011,Y -32.183,Z -59.217,A -90.000,B 90.000,C 0.000} C_DIS
LIN {X -15.745,Y -32.181,Z -59.170,A -90.000,B 90.000,C 0.000} C_DIS
LIN {X -15.610,Y -32.184,Z -59.153,A -90.000,B 90.000,C 0.000} C_DIS
LIN {X -15.260,Y -32.199,Z -59.120,A -90.000,B 90.000,C 0.000} C_DIS
LIN {X -15.152,Y -32.205,Z -59.113,A -90.000,B 90.000,C 0.000} C_DIS
LIN {X -14.458,Y -32.255,Z -59.081,A -90.000,B 90.000,C 0.000} C_DIS
LIN {X -14.215,Y -32.274,Z -59.069,A -90.000,B 90.000,C 0.000} C_DIS
LIN {X -13.777,Y -32.301,Z -59.053,A -90.000,B 90.000,C 0.000} C_DIS
LIN {X -13.326,Y -32.315,Z -59.045,A -90.000,B 90.000,C 0.000} C_DIS
LIN {X -11.862,Y -32.276,Z -59.063,A -90.000,B 90.000,C 0.000} C_DIS
LIN {X -11.722,Y -32.274,Z -59.069,A -90.000,B 90.000,C 0.000} C_DIS
LIN {X -11.371,Y -32.277,Z -59.094,A -90.000,B 90.000,C 0.000} C_DIS
LIN {X -10.948,Y -32.281,Z -59.132,A -90.000,B 90.000,C 0.000} C_DIS
LIN {X -9.821,Y -32.270,Z -59.254,A -90.000,B 90.000,C 0.000} C_DIS
LIN {X -8.627,Y -32.248,Z -59.390,A -90.000,B 90.000,C 0.000} C_DIS
LIN {X -7.715,Y -32.226,Z -59.541,A -90.000,B 90.000,C 0.000} C_DIS
LIN {X -6.513,Y -32.190,Z -59.728,A -90.000,B 90.000,C 0.000} C_DIS
LIN {X -5.946,Y -32.179,Z -59.812,A -90.000,B 90.000,C 0.000} C_DIS
LIN {X -5.243,Y -32.169,Z -59.930,A -90.000,B 90.000,C 0.000} C_DIS
LIN {X -5.109,Y -32.165,Z -59.954,A -90.000,B 90.000,C 0.000} C_DIS
LIN {X -4.350,Y -32.149,Z -60.100,A -90.000,B 90.000,C 0.000} C_DIS
LIN {X -3.270,Y -32.101,Z -60.275,A -90.000,B 90.000,C 0.000} C_DIS
LIN {X -3.139,Y -32.099,Z -60.294,A -90.000,B 90.000,C 0.000} C_DIS
LIN {X -2.728,Y -32.088,Z -60.355,A -90.000,B 90.000,C 0.000} C_DIS
LIN {X -2.533,Y -32.081,Z -60.386,A -90.000,B 90.000,C 0.000} C_DIS
LIN {X -1.839,Y -32.065,Z -60.511,A -90.000,B 90.000,C 0.000} C_DIS
LIN {X -0.807,Y -32.047,Z -60.695,A -90.000,B 90.000,C 0.000} C_DIS
LIN {X -0.234,Y -32.022,Z -60.776,A -90.000,B 90.000,C 0.000} C_DIS
LIN {X 0.018,Y -32.004,Z -60.816,A -90.000,B 90.000,C 0.000} C_DIS
LIN {X 0.901,Y -31.985,Z -60.924,A -90.000,B 90.000,C 0.000} C_DIS
LIN {X 2.077,Y -31.957,Z -61.080,A -90.000,B 90.000,C 0.000} C_DIS
LIN {X 2.690,Y -31.928,Z -61.147,A -90.000,B 90.000,C 0.000} C_DIS
LIN {X 3.082,Y -31.913,Z -61.186,A -90.000,B 90.000,C 0.000} C_DIS
LIN {X 3.530,Y -31.904,Z -61.238,A -90.000,B 90.000,C 0.000} C_DIS
LIN {X 4.779,Y -31.888,Z -61.372,A -90.000,B 90.000,C 0.000} C_DIS
LIN {X 5.049,Y -31.882,Z -61.399,A -90.000,B 90.000,C 0.000} C_DIS
LIN {X 5.246,Y -31.881,Z -61.415,A -90.000,B 90.000,C 0.000} C_DIS
LIN {X 6.774,Y -31.863,Z -61.538,A -90.000,B 90.000,C 0.000} C_DIS
LIN {X 6.980,Y -31.859,Z -61.551,A -90.000,B 90.000,C 0.000} C_DIS
LIN {X 7.985,Y -31.861,Z -61.584,A -90.000,B 90.000,C 0.000} C_DIS
LIN {X 8.513,Y -31.867,Z -61.598,A -90.000,B 90.000,C 0.000} C_DIS
LIN {X 8.614,Y -31.867,Z -61.599,A -90.000,B 90.000,C 0.000} C_DIS
LIN {X 8.856,Y -31.875,Z -61.588,A -90.000,B 90.000,C 0.000} C_DIS
LIN {X 9.776,Y -31.897,Z -61.553,A -90.000,B 90.000,C 0.000} C_DIS
LIN {X 9.839,Y -31.896,Z -61.549,A -90.000,B 90.000,C 0.000} C_DIS
LIN {X 10.043,Y -31.906,Z -61.522,A -90.000,B 90.000,C 0.000} C_DIS
LIN {X 10.540,Y -31.924,Z -61.464,A -90.000,B 90.000,C 0.000} C_DIS
LIN {X 10.750,Y -31.921,Z -61.429,A -90.000,B 90.000,C 0.000} C_DIS
LIN {X 11.045,Y -31.933,Z -61.364,A -90.000,B 90.000,C 0.000} C_DIS
LIN {X 11.284,Y -31.926,Z -61.294,A -90.000,B 90.000,C 0.000} C_DIS
LIN {X 11.474,Y -31.902,Z -61.219,A -90.000,B 90.000,C 0.000} C_DIS
LIN {X 11.521,Y -31.897,Z -61.196,A -90.000,B 90.000,C 0.000} C_DIS
LIN {X 11.867,Y -31.864,Z -61.031,A -90.000,B 90.000,C 0.000} C_DIS
LIN {X 12.291,Y -31.850,Z -60.817,A -90.000,B 90.000,C 0.000} C_DIS
LIN {X 12.505,Y -31.846,Z -60.711,A -90.000,B 90.000,C 0.000} C_DIS
LIN {X 12.781,Y -31.833,Z -60.579,A -90.000,B 90.000,C 0.000} C_DIS
LIN {X 12.984,Y -31.829,Z -60.476,A -90.000,B 90.000,C 0.000} C_DIS
LIN {X 13.217,Y -31.833,Z -60.366,A -90.000,B 90.000,C 0.000} C_DIS
LIN {X 13.319,Y -31.832,Z -60.324,A -90.000,B 90.000,C 0.000} C_DIS
LIN {X 13.590,Y -31.835,Z -60.219,A -90.000,B 90.000,C 0.000} C_DIS
LIN {X 13.765,Y -31.833,Z -60.157,A -90.000,B 90.000,C 0.000} C_DIS
LIN {X 13.881,Y -31.834,Z -60.118,A -90.000,B 90.000,C 0.000} C_DIS
LIN {X 14.170,Y -31.852,Z -60.022,A -90.000,B 90.000,C 0.000} C_DIS
LIN {X 14.259,Y -31.856,Z -59.990,A -90.000,B 90.000,C 0.000} C_DIS
LIN {X 14.457,Y -31.851,Z -59.933,A -90.000,B 90.000,C 0.000} C_DIS
LIN {X 14.671,Y -31.853,Z -59.878,A -90.000,B 90.000,C 0.000} C_DIS
LIN {X 14.945,Y -31.843,Z -59.826,A -90.000,B 90.000,C 0.000} C_DIS
LIN {X 15.045,Y -31.841,Z -59.809,A -90.000,B 90.000,C 0.000} C_DIS
LIN {X 15.110,Y -31.842,Z -59.799,A -90.000,B 90.000,C 0.000} C_DIS
LIN {X 15.296,Y -31.854,Z -59.767,A -90.000,B 90.000,C 0.000} C_DIS
LIN {X 15.508,Y -31.858,Z -59.741,A -90.000,B 90.000,C 0.000} C_DIS
LIN {X 15.712,Y -31.867,Z -59.720,A -90.000,B 90.000,C 0.000} C_DIS
LIN {X 15.778,Y -31.867,Z -59.718,A -90.000,B 90.000,C 0.000} C_DIS
LIN {X 16.134,Y -31.873,Z -59.716,A -90.000,B 90.000,C 0.000} C_DIS
LIN {X 16.320,Y -31.873,Z -59.720,A -90.000,B 90.000,C 0.000} C_DIS
LIN {X 16.734,Y -31.858,Z -59.745,A -90.000,B 90.000,C 0.000} C_DIS
LIN {X 16.873,Y -31.856,Z -59.757,A -90.000,B 90.000,C 0.000} C_DIS
LIN {X 17.188,Y -31.863,Z -59.792,A -90.000,B 90.000,C 0.000} C_DIS
LIN {X 17.355,Y -31.860,Z -59.818,A -90.000,B 90.000,C 0.000} C_DIS
LIN {X 17.526,Y -31.854,Z -59.849,A -90.000,B 90.000,C 0.000} C_DIS
LIN {X 17.732,Y -31.794,Z -59.838,A -90.000,B 90.000,C 0.000} C_DIS
LIN {X 17.915,Y -31.725,Z -59.814,A -90.000,B 90.000,C 0.000} C_DIS
LIN {X 18.007,Y -31.718,Z -59.768,A -90.000,B 90.000,C 0.000} C_DIS
LIN {X 18.237,Y -31.705,Z -59.657,A -90.000,B 90.000,C 0.000} C_DIS
LIN {X 18.466,Y -31.690,Z -59.559,A -90.000,B 90.000,C 0.000} C_DIS
LIN {X 18.491,Y -31.689,Z -59.550,A -90.000,B 90.000,C 0.000} C_DIS
LIN {X 18.779,Y -31.673,Z -59.450,A -90.000,B 90.000,C 0.000} C_DIS
LIN {X 18.893,Y -31.678,Z -59.397,A -90.000,B 90.000,C 0.000} C_DIS
LIN {X 18.955,Y -31.680,Z -59.371,A -90.000,B 90.000,C 0.000} C_DIS
LIN {X 19.201,Y -31.686,Z -59.283,A -90.000,B 90.000,C 0.000} C_DIS
LIN {X 19.469,Y -31.698,Z -59.193,A -90.000,B 90.000,C 0.000} C_DIS
LIN {X 19.575,Y -31.699,Z -59.163,A -90.000,B 90.000,C 0.000} C_DIS
LIN {X 19.839,Y -31.708,Z -59.095,A -90.000,B 90.000,C 0.000} C_DIS
LIN {X 20.270,Y -31.718,Z -59.020,A -90.000,B 90.000,C 0.000} C_DIS
LIN {X 20.397,Y -31.719,Z -59.006,A -90.000,B 90.000,C 0.000} C_DIS
LIN {X 20.844,Y -31.731,Z -58.981,A -90.000,B 90.000,C 0.000} C_DIS
LIN {X 21.017,Y -31.731,Z -58.988,A -90.000,B 90.000,C 0.000} C_DIS
LIN {X 21.283,Y -31.738,Z -59.004,A -90.000,B 90.000,C 0.000} C_DIS
LIN {X 21.418,Y -31.734,Z -59.022,A -90.000,B 90.000,C 0.000} C_DIS
LIN {X 21.522,Y -31.734,Z -59.037,A -90.000,B 90.000,C 0.000} C_DIS
LIN {X 21.730,Y -31.739,Z -59.075,A -90.000,B 90.000,C 0.000} C_DIS
LIN {X 21.758,Y -31.728,Z -59.074,A -90.000,B 90.000,C 0.000} C_DIS
LIN {X 21.946,Y -31.653,Z -59.068,A -90.000,B 90.000,C 0.000} C_DIS
LIN {X 21.990,Y -31.654,Z -59.038,A -90.000,B 90.000,C 0.000} C_DIS
LIN {X 22.270,Y -31.654,Z -58.851,A -90.000,B 90.000,C 0.000} C_DIS
LIN {X 22.546,Y -31.659,Z -58.672,A -90.000,B 90.000,C 0.000} C_DIS
LIN {X 22.754,Y -31.660,Z -58.546,A -90.000,B 90.000,C 0.000} C_DIS
LIN {X 23.083,Y -31.665,Z -58.352,A -90.000,B 90.000,C 0.000} C_DIS
LIN {X 23.567,Y -31.671,Z -58.091,A -90.000,B 90.000,C 0.000} C_DIS
LIN {X 23.987,Y -31.685,Z -57.877,A -90.000,B 90.000,C 0.000} C_DIS
LIN {X 24.323,Y -31.694,Z -57.717,A -90.000,B 90.000,C 0.000} C_DIS
LIN {X 24.478,Y -31.700,Z -57.645,A -90.000,B 90.000,C 0.000} C_DIS
LIN {X 24.593,Y -31.615,Z -57.508,A -90.000,B 90.000,C 0.000} C_DIS
LIN {X 24.664,Y -31.572,Z -57.436,A -90.000,B 90.000,C 0.000} C_DIS
LIN {X 24.773,Y -31.516,Z -57.335,A -90.000,B 90.000,C 0.000} C_DIS
LIN {X 24.869,Y -31.473,Z -57.253,A -90.000,B 90.000,C 0.000} C_DIS
LIN {X 24.940,Y -31.445,Z -57.195,A -90.000,B 90.000,C 0.000} C_DIS
LIN {X 24.925,Y -31.455,Z -56.943,A -90.000,B 90.000,C 0.000} C_DIS
LIN {X 24.918,Y -31.464,Z -56.800,A -90.000,B 90.000,C 0.000} C_DIS
LIN {X 24.926,Y -31.471,Z -56.629,A -90.000,B 90.000,C 0.000} C_DIS
LIN {X 24.940,Y -31.483,Z -56.368,A -90.000,B 90.000,C 0.000} C_DIS
LIN {X 24.941,Y -31.484,Z -56.352,A -90.000,B 90.000,C 0.000} C_DIS
LIN {X 25.008,Y -31.493,Z -55.916,A -90.000,B 90.000,C 0.000} C_DIS
LIN {X 25.123,Y -31.502,Z -55.489,A -90.000,B 90.000,C 0.000} C_DIS
LIN {X 25.155,Y -31.500,Z -55.402,A -90.000,B 90.000,C 0.000} C_DIS
LIN {X 25.276,Y -31.504,Z -55.092,A -90.000,B 90.000,C 0.000} C_DIS
LIN {X 25.310,Y -31.504,Z -55.015,A -90.000,B 90.000,C 0.000} C_DIS
LIN {X 25.339,Y -31.505,Z -54.946,A -90.000,B 90.000,C 0.000} C_DIS
LIN {X 25.420,Y -31.505,Z -54.788,A -90.000,B 90.000,C 0.000} C_DIS
LIN {X 25.538,Y -31.508,Z -54.563,A -90.000,B 90.000,C 0.000} C_DIS
LIN {X 25.705,Y -31.502,Z -54.298,A -90.000,B 90.000,C 0.000} C_DIS
LIN {X 25.786,Y -31.502,Z -54.172,A -90.000,B 90.000,C 0.000} C_DIS
LIN {X 25.841,Y -31.500,Z -54.100,A -90.000,B 90.000,C 0.000} C_DIS
LIN {X 25.997,Y -31.499,Z -53.888,A -90.000,B 90.000,C 0.000} C_DIS
LIN {X 26.030,Y -31.497,Z -53.851,A -90.000,B 90.000,C 0.000} C_DIS
LIN {X 26.091,Y -31.495,Z -53.781,A -90.000,B 90.000,C 0.000} C_DIS
LIN {X 26.307,Y -31.493,Z -53.540,A -90.000,B 90.000,C 0.000} C_DIS
LIN {X 26.468,Y -31.486,Z -53.392,A -90.000,B 90.000,C 0.000} C_DIS
LIN {X 26.651,Y -31.484,Z -53.227,A -90.000,B 90.000,C 0.000} C_DIS
LIN {X 26.819,Y -31.476,Z -53.102,A -90.000,B 90.000,C 0.000} C_DIS
LIN {X 27.024,Y -31.471,Z -52.953,A -90.000,B 90.000,C 0.000} C_DIS
LIN {X 27.109,Y -31.469,Z -52.898,A -90.000,B 90.000,C 0.000} C_DIS
LIN {X 27.363,Y -31.460,Z -52.748,A -90.000,B 90.000,C 0.000} C_DIS
LIN {X 27.530,Y -31.459,Z -52.653,A -90.000,B 90.000,C 0.000} C_DIS
LIN {X 27.728,Y -31.455,Z -52.549,A -90.000,B 90.000,C 0.000} C_DIS
LIN {X 27.741,Y -31.468,Z -52.508,A -90.000,B 90.000,C 0.000} C_DIS
LIN {X 27.786,Y -31.510,Z -52.378,A -90.000,B 90.000,C 0.000} C_DIS
LIN {X 27.830,Y -31.553,Z -52.262,A -90.000,B 90.000,C 0.000} C_DIS
LIN {X 27.926,Y -31.632,Z -52.065,A -90.000,B 90.000,C 0.000} C_DIS
LIN {X 27.954,Y -31.656,Z -52.011,A -90.000,B 90.000,C 0.000} C_DIS
LIN {X 28.034,Y -31.726,Z -51.871,A -90.000,B 90.000,C 0.000} C_DIS
LIN {X 28.072,Y -31.757,Z -51.814,A -90.000,B 90.000,C 0.000} C_DIS
LIN {X 28.131,Y -31.761,Z -51.532,A -90.000,B 90.000,C 0.000} C_DIS
LIN {X 28.181,Y -31.758,Z -51.320,A -90.000,B 90.000,C 0.000} C_DIS
LIN {X 28.296,Y -31.757,Z -50.864,A -90.000,B 90.000,C 0.000} C_DIS
LIN {X 28.326,Y -31.753,Z -50.776,A -90.000,B 90.000,C 0.000} C_DIS
LIN {X 28.377,Y -31.751,Z -50.640,A -90.000,B 90.000,C 0.000} C_DIS
LIN {X 28.424,Y -31.751,Z -50.518,A -90.000,B 90.000,C 0.000} C_DIS
LIN {X 28.495,Y -31.749,Z -50.339,A -90.000,B 90.000,C 0.000} C_DIS
LIN {X 28.573,Y -31.748,Z -50.153,A -90.000,B 90.000,C 0.000} C_DIS
LIN {X 28.690,Y -31.750,Z -49.885,A -90.000,B 90.000,C 0.000} C_DIS
LIN {X 28.810,Y -31.743,Z -49.646,A -90.000,B 90.000,C 0.000} C_DIS
LIN {X 28.910,Y -31.742,Z -49.455,A -90.000,B 90.000,C 0.000} C_DIS
LIN {X 29.075,Y -31.729,Z -49.181,A -90.000,B 90.000,C 0.000} C_DIS
LIN {X 29.139,Y -31.727,Z -49.080,A -90.000,B 90.000,C 0.000} C_DIS
LIN {X 29.258,Y -31.730,Z -48.895,A -90.000,B 90.000,C 0.000} C_DIS
LIN {X 29.419,Y -31.731,Z -48.655,A -90.000,B 90.000,C 0.000} C_DIS
LIN {X 29.521,Y -31.735,Z -48.510,A -90.000,B 90.000,C 0.000} C_DIS
LIN {X 29.705,Y -31.726,Z -48.283,A -90.000,B 90.000,C 0.000} C_DIS
LIN {X 29.794,Y -31.720,Z -48.172,A -90.000,B 90.000,C 0.000} C_DIS
LIN {X 29.856,Y -31.713,Z -48.105,A -90.000,B 90.000,C 0.000} C_DIS
LIN {X 30.193,Y -31.687,Z -47.762,A -90.000,B 90.000,C 0.000} C_DIS
LIN {X 30.282,Y -31.687,Z -47.669,A -90.000,B 90.000,C 0.000} C_DIS
LIN {X 30.548,Y -31.687,Z -47.419,A -90.000,B 90.000,C 0.000} C_DIS
LIN {X 30.616,Y -31.686,Z -47.356,A -90.000,B 90.000,C 0.000} C_DIS
LIN {X 30.994,Y -31.678,Z -47.065,A -90.000,B 90.000,C 0.000} C_DIS
LIN {X 31.222,Y -31.663,Z -46.908,A -90.000,B 90.000,C 0.000} C_DIS
LIN {X 31.359,Y -31.652,Z -46.821,A -90.000,B 90.000,C 0.000} C_DIS
LIN {X 31.723,Y -31.620,Z -46.611,A -90.000,B 90.000,C 0.000} C_DIS
LIN {X 32.130,Y -31.608,Z -46.396,A -90.000,B 90.000,C 0.000} C_DIS
LIN {X 32.278,Y -31.603,Z -46.323,A -90.000,B 90.000,C 0.000} C_DIS
LIN {X 32.481,Y -31.604,Z -46.229,A -90.000,B 90.000,C 0.000} C_DIS
LIN {X 32.547,Y -31.602,Z -46.203,A -90.000,B 90.000,C 0.000} C_DIS
LIN {X 32.900,Y -31.593,Z -46.069,A -90.000,B 90.000,C 0.000} C_DIS
LIN {X 33.392,Y -31.565,Z -45.924,A -90.000,B 90.000,C 0.000} C_DIS
LIN {X 33.572,Y -31.551,Z -45.882,A -90.000,B 90.000,C 0.000} C_DIS
LIN {X 33.792,Y -31.541,Z -45.834,A -90.000,B 90.000,C 0.000} C_DIS
LIN {X 34.012,Y -31.528,Z -45.791,A -90.000,B 90.000,C 0.000} C_DIS
LIN {X 34.261,Y -31.518,Z -45.746,A -90.000,B 90.000,C 0.000} C_DIS
LIN {X 34.545,Y -31.512,Z -45.688,A -90.000,B 90.000,C 0.000} C_DIS
LIN {X 34.699,Y -31.512,Z -45.658,A -90.000,B 90.000,C 0.000} C_DIS
LIN {X 34.820,Y -31.515,Z -45.635,A -90.000,B 90.000,C 0.000} C_DIS
LIN {X 35.007,Y -31.511,Z -45.618,A -90.000,B 90.000,C 0.000} C_DIS
LIN {X 35.280,Y -31.509,Z -45.593,A -90.000,B 90.000,C 0.000} C_DIS
LIN {X 35.616,Y -31.505,Z -45.572,A -90.000,B 90.000,C 0.000} C_DIS
LIN {X 35.824,Y -31.500,Z -45.559,A -90.000,B 90.000,C 0.000} C_DIS
LIN {X 36.040,Y -31.488,Z -45.562,A -90.000,B 90.000,C 0.000} C_DIS
LIN {X 36.213,Y -31.477,Z -45.567,A -90.000,B 90.000,C 0.000} C_DIS
LIN {X 36.558,Y -31.463,Z -45.580,A -90.000,B 90.000,C 0.000} C_DIS
LIN {X 36.796,Y -31.452,Z -45.595,A -90.000,B 90.000,C 0.000} C_DIS
LIN {X 37.117,Y -31.444,Z -45.619,A -90.000,B 90.000,C 0.000} C_DIS
LIN {X 37.286,Y -31.439,Z -45.635,A -90.000,B 90.000,C 0.000} C_DIS
LIN {X 37.563,Y -31.437,Z -45.663,A -90.000,B 90.000,C 0.000} C_DIS
LIN {X 37.953,Y -31.430,Z -45.721,A -90.000,B 90.000,C 0.000} C_DIS
LIN {X 38.822,Y -31.423,Z -45.847,A -90.000,B 90.000,C 0.000} C_DIS
LIN {X 39.069,Y -31.424,Z -45.884,A -90.000,B 90.000,C 0.000} C_DIS
LIN {X 39.203,Y -31.426,Z -45.901,A -90.000,B 90.000,C 0.000} C_DIS
LIN {X 40.146,Y -31.457,Z -46.025,A -90.000,B 90.000,C 0.000} C_DIS
LIN {X 40.793,Y -31.505,Z -46.053,A -90.000,B 90.000,C 0.000} C_DIS
LIN {X 41.128,Y -31.552,Z -46.019,A -90.000,B 90.000,C 0.000} C_DIS
LIN {X 41.578,Y -31.622,Z -45.978,A -90.000,B 90.000,C 0.000} C_DIS
LIN {X 41.653,Y -31.637,Z -45.968,A -90.000,B 90.000,C 0.000} C_DIS
